RoboDK station: invisiblechess.rdk

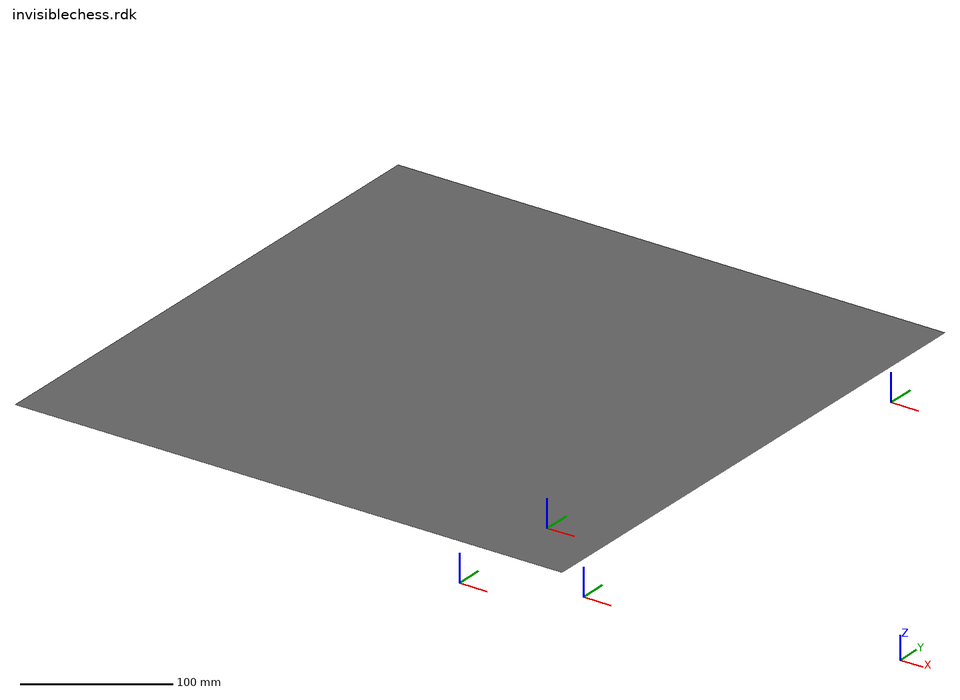
[picture v0: the station drawn from its stored meshes, robots at their saved joint values, targets as dots, program paths as lines]
Station invisiblechess (saved by RoboDK 5.6.5). Poses are relative to the parent item; angles as X-Y-Z fixed-axis rotations.
Station parameters (name, value as stored): Record_Record, 0
  - frame Frame 1 at (0, -100, 0) mm
    - object chessrobo at (100, -100, -10) mm, size 437.3 x 437.3 x 0 mm, 469029088 curves, geometry from chessrobo.png
    - object PAWN at (65, 300, -10) mm
    - object KNIGHT at (117, 146, -10) mm
    - object bishop at (-185, 150, -10) mm
    - object PAWN at (17, 96, -10) mm
    - object KNIGHT at (115, 300, -10) mm
    - object bishop at (17, 96, -10) mm
    - object PAWN at (67, 146, -10) mm
    - object KNIGHT at (-35, 200, -10) mm
    - object king at (67, 196, -10) mm
  - frame Frame 3 at (67, -54, -10) mm
    - object bishop at (0, 0, 0) mm
    - object PAWN at (0, 0, 0) mm
    - object ROOK at (-200, 0, 0) mm
    - object KNIGHT at (0, 0, 0) mm
    - object ROOK at (-200, 0, 0) mm
    - object PAWN at (0, 0, 0) mm
    - object PAWN at (0, 0, 0) mm
    - object PAWN at (0, 0, 0) mm
    - object PAWN at (0, 0, 0) mm
    - object QUEEN at (0, 0, 0) mm
    - object PAWN at (0, 0, 0) mm
  - Python program chess1 (listed below)
  - program rookie (3 instructions, listed below)
  - program backtobse (1 instructions, listed below)
  - frame Frame 4 at (0, 0, 0) mm
    - frame Frame 3 at (65, 300, -10) mm
      - object ROOK at (-200, 0, 0) mm
      - object king at (0, 0, 0) mm
      - object QUEEN at (0, 0, 0) mm
      - object ROOK at (-200, 0, 0) mm
      - object bishop at (0, 0, 0) mm
      - object PAWN at (0, 0, 0) mm
      - object PAWN at (0, 0, 0) mm
      - object PAWN at (0, 0, 0) mm
      - object PAWN at (0, 0, 0) mm
      - object PAWN at (0, 0, 0) mm
      - object PAWN at (0, 0, 0) mm
      - object PAWN at (0, 0, 0) mm
  - Python program Prog4 (listed below)
  - Python program chess (listed below)
  - program Prog6 (1 instructions, listed below)
  - program Prog7 (1 instructions, listed below)
  - program Prog8 (1 instructions, listed below)
  - program Prog9 (0 instructions, listed below)
  - program Prog10 (0 instructions, listed below)
  - Python program Prog11 (listed below)
  - Python program samattach (listed below)
  - Python program Prog13 (listed below)
  - Python program Prog14 (listed below)
  - Python program Prog15 (listed below)
  - Python program Prog16 (listed below)
  - frame My Mechanism Base at (0, 0, 0) mm
    - robot My Mechanism: 4 axes
        joint limits [-2000, -2000, -2000, -2000] to [2000, 2000, 2000, 2000]; home [0, 0, 0, 0]; saved at [-150, 150, -10, 0]
      - tool microagv1, TCP at (0, 0, 0) mm
  - Python program Prog17 (listed below)
  - Python program Prog18 (listed below)
  - Python program Prog19 (listed below)
  - Python program Prog20 (listed below)
  - Python program Prog21 (listed below)
  - Python program Prog22 (listed below)
  - Python program final (listed below)
  - Python program Prog24 (listed below)
  - Python program Prog25 (listed below)
  - frame Frame 6 at (-200, 150, 1000) mm, rotated rx 180 ry 0 rz -90 deg
    - camera Camera 1
  - Python program app (listed below)
  - Python program code (listed below)
  - Python program code (listed below)
  - Python program Prog29 (listed below)
  - frame Frame 7 at (0, 1150, 0) mm
  - Python program chessmaster1 (listed below)
  - Python program Prog31 (listed below)
  - Python program Prog32 (listed below)
  - Python program Prog33 (listed below)
  - Python program Prog34 (listed below)
  - Python program Prog35 (listed below)
  - Python program Prog36 (listed below)
  - Python program final (listed below)
  - Python program stockfish (listed below)
  - Python program RoboDKChessStockfishfinal (listed below)

--- Python program chess1 ---
# Type help("robodk.robolink") or help("robodk.robomath") for more information
# Press F5 to run the script
# Documentation: https://robodk.com/doc/en/RoboDK-API.html
# Reference:     https://robodk.com/doc/en/PythonAPI/robodk.html
# Note: It is not required to keep a copy of this file, your Python script is saved with your RDK project

# You can also use the new version of the API:
from robodk import robolink    # RoboDK API
from robodk import robomath    # Robot toolbox
RDK = robolink.Robolink()

# Forward and backwards compatible use of the RoboDK API:
# Remove these 2 lines to follow python programming guidelines
from robodk import *      # RoboDK API
from robolink import *    # Robot toolbox
# Link to RoboDK
# RDK = Robolink()

# Notify user:
print('To edit this program:\nright click on the Python program, then, select "Edit Python script"')

# Program example:

# Provoking an exception will display the console output if you run this script from RoboDK
#raise Exception('Program not edited.')
item = RDK.Item('My Mechanism')
if item.Valid():
    print('Item selected: ' + item.Name())
    print('Item position before move: ' + repr(item.Pose()))

def move_rook1():
    current_pose = item.Pose()
    new_pose = transl(-350, 0, 0) * current_pose
    item.MoveL(new_pose)

def move_rook2():
    current_pose = item.Pose()
    new_pose = transl(0, 350, 0) * current_pose
    item.MoveL(new_pose)

def move_rook3():
    current_pose = item.Pose()
    new_pose = transl(350, 0, 0) * current_pose
    item.MoveL(new_pose)

def move_rook4():
    current_pose = item.Pose()
    new_pose = transl(0, -350, 0) * current_pose
    item.MoveL(new_pose)

move_rook1()
move_rook2()
move_rook3()
move_rook4()

--- program rookie ---
  Attach to microagv1
  Call chess
  Detach from AGV

--- program backtobse ---
  Replace ROOK

--- Python program Prog4 ---
# Type help("robodk.robolink") or help("robodk.robomath") for more information
# Press F5 to run the script
# Documentation: https://robodk.com/doc/en/RoboDK-API.html
# Reference:     https://robodk.com/doc/en/PythonAPI/robodk.html
# Note: It is not required to keep a copy of this file, your Python script is saved with your RDK project

# You can also use the new version of the API:
from robodk import robolink    # RoboDK API
from robodk import robomath    # Robot toolbox
RDK = robolink.Robolink()

# Forward and backwards compatible use of the RoboDK API:
# Remove these 2 lines to follow python programming guidelines
from robodk import *      # RoboDK API
from robolink import *    # Robot toolbox
# Link to RoboDK
# RDK = Robolink()

# Notify user:
print('To edit this program:\nright click on the Python program, then, select "Edit Python script"')

# Program example:
item = RDK.Item('base')
if item.Valid():
    print('Item selected: ' + item.Name())
    print('Item posistion: ' + repr(item.Pose()))

print('Items in the station:')
itemlist = RDK.ItemList()
print(itemlist)

# Provoking an exception will display the console output if you run this script from RoboDK
#raise Exception('Program not edited.')
from robodk import robolink, transl

RDK = robolink.Robolink()

item = RDK.Item('My Mechanism')
if item.Valid():
    print('Item selected: ' + item.Name())
    print('Item position before move: ' + repr(item.Pose()))

# Define the grid and corresponding coordinates
grid_coordinates = {
    'a1': [0, 350, 0],
    'a2': [0, 300, 0],
    'a3': [-350, 350, 0],
    'a4': [-350, 700, 0],
    'a5': [-350, 1050, 0],
    'a6': [-350, 1400, 0],
    'a7': [-350, 1750, 0],
    'a8': [-350, 2100, 0],
    # Add similar entries for b1, c1, etc.
}

def move_to_square(square):
    if square in grid_coordinates:
        current_pose = item.Pose()
        new_pose = transl(*grid_coordinates[square]) * current_pose
        item.MoveL(new_pose)
    else:
        print(f"Square {square} not found in the grid_coordinates dictionary.")

# Prompt the user for input
#target_square = input("Enter the target square (e.g., a1, b3, h8): ")
#move_to_square(target_square)

while True:
    target_square = input("Enter the target square (e.g., a1, b3, h8) or 'no' to exit: ")

    if target_square.lower() == 'no':
        print("Exiting the program.")
        break  # Exit the loop if the user enters 'no'

    move_to_square(target_square)

--- Python program chess ---
from robodk import robolink    # RoboDK API
from robodk import robomath    # Robot toolbox
RDK = robolink.Robolink()

# Forward and backwards compatible use of the RoboDK API:
# Remove these 2 lines to follow python programming guidelines
from robodk import *      # RoboDK API
from robolink import *    # Robot toolbox
from robodk import robolink, transl
RDK = robolink.Robolink()

item = RDK.Item('My Mechanism')
tool = RDK.Item('AGV')
if item.Valid():
    print('Item selected: ' + item.Name())
    print('Item position before move: ' + repr(item.Pose()))
obj = RDK.Item('')
# Define the grid and corresponding coordinates
grid_coordinates = {
    'a1': [0, 350, -10],
    'a2': [0, 300, -10],
    'a3': [0, 250, -10],
    'a4': [0, 200, -10],
    'a5': [0, 150, -10],
    'a6': [0, 100, -10],
    'a7': [0, 50, -10],
    'a8': [0, 0, -10],
    'b1': [-50, 350, -10],
    'b2': [-50, 300, -10],
    'b3': [-50, 250, -10],
    'b4': [-50, 200, -10],
    'b5': [-50, 150, -10],
    'b6': [-50, 100, -10],
    'b7': [-50, 50, -10],
    'b8': [-50, 0, -10],
    'c1': [-100, 350, -10],
    'c2': [-100, 300, -10],
    'c3': [-100, 250, -10],
    'c4': [-100, 200, -10],
    'c5': [-100, 150, -10],
    'c6': [-100, 100, -10],
    'c7': [-100, 50, -10],
    'c8': [-100, 0, -10],
    'd1': [-150, 350, -10],
    'd2': [-150, 300, -10],
    'd3': [-150, 250, -10],
    'd4': [-150, 200, -10],
    'd5': [-150, 150, -10],
    'd6': [-150, 100, -10],
    'd7': [-150, 50, -10],
    'd8': [-150, 0, -10],
    'e1': [-200, 350, -10],
    'e2': [-200, 300, -10],
    'e3': [-200, 250, -10],
    'e4': [-200, 200, -10],
    'e5': [-200, 150, -10],
    'e6': [-200, 100, -10],
    'e7': [-200, 50, -10],
    'e8': [-200, 0, -10],
    'f1': [-250, 350, -10],
    'f2': [-250, 300, -10],
    'f3': [-250, 250, -10],
    'f4': [-250, 200, -10],
    'f5': [-250, 150, -10],
    'f6': [-250, 100, -10],
    'f7': [-250, 50, -10],
    'f8': [-250, 0, -10],
    'g1': [-300, 350, -10],
    'g2': [-300, 300, -10],
    'g3': [-300, 250, -10],
    'g4': [-300, 200, -10],
    'g5': [-300, 150, -10],
    'g6': [-300, 100, -10],
    'g7': [-300, 50, -10],
    'g8': [-300, 0, -10],
    'h1': [-350, 350, -10],
    'h2': [-350, 300, -10],
    'h3': [-350, 250, -10],
    'h4': [-350, 200, -10],
    'h5': [-350, 150, -10],
    'h6': [-350, 100, -10],
    'h7': [-350, 50, -10],
    'h8': [-350, 0, -10],
}

def move_to_square(square):
    if square in grid_coordinates:
        target_pose = transl(*grid_coordinates[square])
        item.setPose(target_pose)  # Set the robot's pose directly
    else:
        print(f"Square {square} not found in the grid_coordinates dictionary.")




# Loop to keep asking for input
while True:
    target_square = input("Enter the target square (e.g., a1, b3, h8) or 'no' to exit: ")

    if target_square.lower() == 'no':
        print("Exiting the program.")
        break  # Exit the loop if the user enters 'no'

    move_to_square(target_square)
    #tool.AttachClosest(list_objects=[obj])
    tool.RDK().RunProgram('Prog7')
    target_square = input("Enter the target square (e.g., a1, b3, h8) or 'no' to exit: ")

    if target_square.lower() == 'no':
        print("Exiting the program.")
        break  # Exit the loop if the user enters 'no'

    move_to_square(target_square)
    tool.RDK().RunProgram('Prog8')

--- program Prog6 ---
  Replace objects

--- program Prog7 ---
  Attach to microagv1

--- program Prog8 ---
  Detach from microagv1

--- program Prog9 ---

--- program Prog10 ---

--- Python program Prog11 ---
# Type help("robodk.robolink") or help("robodk.robomath") for more information
# Press F5 to run the script
# Documentation: https://robodk.com/doc/en/RoboDK-API.html
# Reference:     https://robodk.com/doc/en/PythonAPI/robodk.html
# Note: It is not required to keep a copy of this file, your Python script is saved with your RDK project

# You can also use the new version of the API:
from robodk import robolink    # RoboDK API
from robodk import robomath    # Robot toolbox
RDK = robolink.Robolink()

# Forward and backwards compatible use of the RoboDK API:
# Remove these 2 lines to follow python programming guidelines
from robodk import *      # RoboDK API
from robolink import *    # Robot toolbox
# Link to RoboDK
# RDK = Robolink()
from robodk import robolink, robomath
# Notify user:
print('To edit this program:\nright click on the Python program, then, select "Edit Python script"')

# Program example:
item = RDK.Item('My Mechanism')
if item.Valid():
    print('Item selected: ' + item.Name())
    print('Item posistion: ' + repr(item.Pose()))

print('Items in the station:')
itemlist = RDK.ItemList()
print(itemlist)

# Provoking an exception will display the console output if you run this script from RoboDK
#raise Exception('Program not edited.')
from robodk import robolink, transl
from robodk import robolink, robomath
RDK = robolink.Robolink()

# This will automatically select the robot if there is only one
robot = RDK.ItemUserPick("", robolink.ITEM_TYPE_ROBOT_ARM)
if not robot.Valid():
    quit()
RDK = robolink.Robolink()

item = RDK.Item('My Mechanism')
if item.Valid():
    print('Item selected: ' + item.Name())
    print('Item position before move: ' + repr(item.Pose()))

# Define the grid and corresponding coordinates
grid_coordinates = {
    'a1': [0, 350, 0],
    'a2': [0, 300, 0],
    'a3': [0, 250, 0],
    'a4': [0, 200, 0],
    'a5': [0, 150, 0],
    'a6': [0, 100, 0],
    'a7': [0, 50, 0],
    'a8': [0, 0, 0],
    # Add similar entries for b1, c1, etc.
}
# Retrieve the active tool of the robot
tool = RDK.getLink(robolink.ITEM_TYPE_TOOL)
if not tool.Valid():
    quit()

# Get the knight object and its current parent (to restore it later)
obj = RDK.Item('')
parent = obj.Parent()  # IMPORTANT! Parent must be a FRAME, not a folder..
def move_to_square(square):
    if square in grid_coordinates:
        target_pose = transl(*grid_coordinates[square])
        item.setPose(target_pose)  # Set the robot's pose directly

        # Attach the closest part on the first move
        closest_part = item.AttachClosest()
        if closest_part.Valid():
            print(f"Attached closest part: {closest_part.Name()}")

        # Detach on the second move
        second_move = input("Enter 'no' to exit or press Enter to make the second move: ")
        if second_move.lower() == 'no':
            print("Exiting the program.")
            return

        item.DetachAll()
        print("Detached all parts.")
    else:
        print(f"Square {square} not found in the grid_coordinates dictionary.")

# Loop to keep asking for input
while True:
    target_square = input("Enter the target square (e.g., a1, b3, h8) or 'no' to exit: ")

    if target_square.lower() == 'no':
        print("Exiting the program.")
        break  # Exit the loop if the user enters 'no'

    move_to_square(target_square)

--- Python program samattach ---
from robodk import robolink, robomath
RDK = robolink.Robolink()

# This will automatically select the robot if there is only one
robot = RDK.ItemUserPick("", robolink.ITEM_TYPE_ROBOT_ARM)
if not robot.Valid():
    quit()

# Retrieve the active tool of the robot
tool = robot.getLink(robolink.ITEM_TYPE_TOOL)
if not tool.Valid():
    quit()

# Get the knight object and its current parent (to restore it later)
obj = RDK.Item('KNIGHT W 1')
parent = obj.Parent() # IMPROTANT! Parent must be a FRAME, not a folder..

robot.MoveJ(RDK.Item('App Pick'))
robot.MoveL(RDK.Item('Pick'))

# In Tools-Options-Station -> check "Check shorted distance between TCP and object shape"
tool.AttachClosest(list_objects=[obj])

robot.MoveL(RDK.Item('App Pick'))
robomath.pause(2)
robot.MoveL(RDK.Item('Pick'))
tool.DetachAll(parent)
robot.MoveL(RDK.Item('App Pick'))

--- Python program Prog13 ---
# Type help("robodk.robolink") or help("robodk.robomath") for more information
# Press F5 to run the script
# Documentation: https://robodk.com/doc/en/RoboDK-API.html
# Reference:     https://robodk.com/doc/en/PythonAPI/robodk.html
# Note: It is not required to keep a copy of this file, your Python script is saved with your RDK project

# You can also use the new version of the API:
from robodk import robolink    # RoboDK API
from robodk import robomath    # Robot toolbox
RDK = robolink.Robolink()

# Forward and backwards compatible use of the RoboDK API:
# Remove these 2 lines to follow python programming guidelines
from robodk import *      # RoboDK API
from robolink import *    # Robot toolbox
# Link to RoboDK
# RDK = Robolink()

# Notify user:
print('To edit this program:\nright click on the Python program, then, select "Edit Python script"')

# Program example:
item = RDK.Item('base')
if item.Valid():
    print('Item selected: ' + item.Name())
    print('Item posistion: ' + repr(item.Pose()))

print('Items in the station:')
itemlist = RDK.ItemList()
print(itemlist)

# Provoking an exception will display the console output if you run this script from RoboDK
raise Exception('Program not edited.')

--- Python program Prog14 ---
from robodk import robolink, ITEM_TYPE_ROBOT_ARM

RDK = robolink.Robolink()

# Retrieve the robot if there is only one
robot = RDK.ItemUserPick("Select a robot", ITEM_TYPE_ROBOT_ARM)
if not robot.Valid():
    quit()

# Retrieve the active tool of the robot
tool = robot.Child()
if not tool.Valid():
    quit()

# Define the grid and corresponding coordinates
grid_coordinates = {
    'a1': [0, 350, 0],
    'a2': [0, 300, 0],
    'a3': [0, 250, 0],
    'a4': [0, 200, 0],
    'a5': [0, 150, 0],
    'a6': [0, 100, 0],
    'a7': [0, 50, 0],
    'a8': [0, 0, 0],
    # Add similar entries for b1, c1, etc.
}

def move_to_square(square):
    if square in grid_coordinates:
        target_pose = robolink.transl(*grid_coordinates[square])
        robot.setPose(target_pose)  # Set the robot's pose directly
        return True
    else:
        print(f"Square {square} not found in the grid_coordinates dictionary.")
        return False

# Variables to keep track of the state
attached = False

# Loop to keep asking for input
while True:
    target_square = input("Enter the target square (e.g., a1, b3, h8) or 'no' to exit: ")

    if target_square.lower() == 'no':
        print("Exiting the program.")
        break  # Exit the loop if the user enters 'no'

    if attached:
        tool.DetachAll()
        print("Detached part.")
        attached = False
    else:
        success = move_to_square(target_square)
        if success:
            tool.AttachClosest()
            print("Attached closest part.")
            attached = True

--- Python program Prog15 ---
# Type help("robodk.robolink") or help("robodk.robomath") for more information
# Press F5 to run the script
# Documentation: https://robodk.com/doc/en/RoboDK-API.html
# Reference:     https://robodk.com/doc/en/PythonAPI/robodk.html
# Note: It is not required to keep a copy of this file, your Python script is saved with your RDK project

# You can also use the new version of the API:
from robodk import robolink    # RoboDK API
from robodk import robomath    # Robot toolbox
RDK = robolink.Robolink()

# Forward and backwards compatible use of the RoboDK API:
# Remove these 2 lines to follow python programming guidelines
from robodk import *      # RoboDK API
from robolink import *    # Robot toolbox
# Link to RoboDK
# RDK = Robolink()

# Notify user:
print('To edit this program:\nright click on the Python program, then, select "Edit Python script"')

# Program example:
item = RDK.Item('base')
if item.Valid():
    print('Item selected: ' + item.Name())
    print('Item posistion: ' + repr(item.Pose()))

print('Items in the station:')
itemlist = RDK.ItemList()
print(itemlist)

# Provoking an exception will display the console output if you run this script from RoboDK
#raise Exception('Program not edited.')
from robodk import *

RDK = robolink.Robolink()

# Retrieve the robot if there is only one
robot = RDK.ItemUserPick("Select a robot", ITEM_TYPE_ROBOT_ARM)
if not robot.Valid():
    quit()

# Retrieve the active tool of the robot
tool = robot.Child()
if not tool.Valid():
    quit()

# Define the grid and corresponding coordinates
grid_coordinates = {
    'a1': [0, 350, 0],
    'a2': [0, 300, 0],
    'a3': [0, 250, 0],
    'a4': [0, 200, 0],
    'a5': [0, 150, 0],
    'a6': [0, 100, 0],
    'a7': [0, 50, 0],
    'a8': [0, 0, 0],
    # Add similar entries for b1, c1, etc.
}

def move_to_square(square):
    if square in grid_coordinates:
        target_pose = transl(*grid_coordinates[square])
        robot.setPose(target_pose)  # Set the robot's pose directly
        return True
    else:
        print(f"Square {square} not found in the grid_coordinates dictionary.")
        return False

# Variables to keep track of the state
attached = False

# Loop to keep asking for input
while True:
    target_square = input("Enter the target square (e.g., a1, b3, h8) or 'no' to exit: ")

    if target_square.lower() == 'no':
        print("Exiting the program.")
        break  # Exit the loop if the user enters 'no'

    if attached:
        tool.DetachAll()
        print("Detached part.")
        attached = False
    else:
        success = move_to_square(target_square)
        if success:
            tool.AttachClosest()
            print("Attached closest part.")
            attached = True

--- Python program Prog16 ---
# Type help("robodk.robolink") or help("robodk.robomath") for more information
# Press F5 to run the script
# Documentation: https://robodk.com/doc/en/RoboDK-API.html
# Reference:     https://robodk.com/doc/en/PythonAPI/robodk.html
# Note: It is not required to keep a copy of this file, your Python script is saved with your RDK project

# You can also use the new version of the API:
from robodk import robolink    # RoboDK API
from robodk import robomath    # Robot toolbox
RDK = robolink.Robolink()

# Forward and backwards compatible use of the RoboDK API:
# Remove these 2 lines to follow python programming guidelines
from robodk import *      # RoboDK API
from robolink import *    # Robot toolbox
# Link to RoboDK
# RDK = Robolink()

# Notify user:
print('To edit this program:\nright click on the Python program, then, select "Edit Python script"')

# Program example:
item = RDK.Item('base')
if item.Valid():
    print('Item selected: ' + item.Name())
    print('Item posistion: ' + repr(item.Pose()))

print('Items in the station:')
itemlist = RDK.ItemList()
print(itemlist)

# Provoking an exception will display the console output if you run this script from RoboDK
#raise Exception('Program not edited.')
from robodk import robolink, transl
import chess
import chess.engine

RDK = robolink.Robolink()

item = RDK.Item('My Mechanism')
tool = RDK.Item('AGV')
if item.Valid():
    print('Item selected: ' + item.Name())
    print('Item position before move: ' + repr(item.Pose()))
obj = RDK.Item('')
# Define the grid and corresponding coordinates
grid_coordinates = {
    'a1': [0, 350, 10],
    'a2': [0, 300, 10],
    'a3': [0, 250, 10],
    'a4': [0, 200, 10],
    'a5': [0, 150, 10],
    'a6': [0, 100, 10],
    'a7': [0, 50, 10],
    'a8': [0, 0, 10],
    # Add similar entries for b1, c1, etc.
}

def move_to_square(square):
    if square in grid_coordinates:
        target_pose = transl(*grid_coordinates[square])
        item.setPose(target_pose)  # Set the robot's pose directly
    else:
        print(f"Square {square} not found in the grid_coordinates dictionary.")

def stockfish_move(board):
    with chess.engine.SimpleEngine.popen_uci("/path/to/stockfish") as engine:
        result = engine.play(board, chess.engine.Limit(time=2.0))
        return result.move

# Loop to keep asking for input
while True:
    target_square = input("Enter the target square (e.g., a1, b3, h8) or 'no' to exit: ")

    if target_square.lower() == 'no':
        print("Exiting the program.")
        break  # Exit the loop if the user enters 'no'

    move_to_square(target_square)
    tool.RDK().RunProgram('Prog7')

    board = chess.Board()
    opponent_move = stockfish_move(board)
    print("Opponent's move:", opponent_move.uci())

    # Assuming opponent_move.uci() returns a valid square (e.g., "e2e4")
    move_to_square(opponent_move.uci())
    tool.RDK().RunProgram('Prog8')

--- Python program Prog17 ---
# Type help("robodk.robolink") or help("robodk.robomath") for more information
# Press F5 to run the script
# Documentation: https://robodk.com/doc/en/RoboDK-API.html
# Reference:     https://robodk.com/doc/en/PythonAPI/robodk.html
# Note: It is not required to keep a copy of this file, your Python script is saved with your RDK project

# You can also use the new version of the API:
from robodk import robolink    # RoboDK API
from robodk import robomath    # Robot toolbox
RDK = robolink.Robolink()

# Forward and backwards compatible use of the RoboDK API:
# Remove these 2 lines to follow python programming guidelines
from robodk import *      # RoboDK API
from robolink import *    # Robot toolbox
# Link to RoboDK
# RDK = Robolink()

# Notify user:
print('To edit this program:\nright click on the Python program, then, select "Edit Python script"')

# Program example:
item = RDK.Item('base')
if item.Valid():
    print('Item selected: ' + item.Name())
    print('Item posistion: ' + repr(item.Pose()))

print('Items in the station:')
itemlist = RDK.ItemList()
print(itemlist)

# Provoking an exception will display the console output if you run this script from RoboDK
#raise Exception('Program not edited.')
import chess
from serial.tools import list_ports
#import chess.svg
import chess.engine
def main():
    # Specify the full path to your Stockfish executable
    engine_path = "stockfish\stockfish-windows-x86-64-avx2"  # Replace with the actual name of your Stockfish executable

    # Create a Chess engine with Stockfish
    engine = chess.engine.SimpleEngine.popen_uci(engine_path)

    board = chess.Board()

--- Python program Prog18 ---
# Type help("robodk.robolink") or help("robodk.robomath") for more information
# Press F5 to run the script
# Documentation: https://robodk.com/doc/en/RoboDK-API.html
# Reference:     https://robodk.com/doc/en/PythonAPI/robodk.html
# Note: It is not required to keep a copy of this file, your Python script is saved with your RDK project

# You can also use the new version of the API:
from robodk import robolink    # RoboDK API
from robodk import robomath    # Robot toolbox
RDK = robolink.Robolink()

# Forward and backwards compatible use of the RoboDK API:
# Remove these 2 lines to follow python programming guidelines
from robodk import *      # RoboDK API
from robolink import *    # Robot toolbox
# Link to RoboDK
# RDK = Robolink()

# Notify user:
#print('To edit this program:\nright click on the Python program, then, select "Edit Python script"')

# Program example:
item = RDK.Item('base')
if item.Valid():
    print('Item selected: ' + item.Name())
    print('Item posistion: ' + repr(item.Pose()))

print('Items in the station:')
itemlist = RDK.ItemList()
#print(itemlist)

# Provoking an exception will display the console output if you run this script from RoboDK
#raise Exception('Program not edited.')
from robolink import import_install
import_install("chess")
import chess
from robolink import import_install
import_install("stockfish")
import stockfish
from stockfish import Stockfish

stockfish = Stockfish(path= "/Users/dancr/chess-robot/stockfish/stockfish-windows-x86-64-avx2.exe")
boardmac = stockfish.get_board_visual()
boardmaco = stockfish.get_best_move()
print(boardmac)
print(boardmaco)

--- Python program Prog19 ---
# Type help("robodk.robolink") or help("robodk.robomath") for more information
# Press F5 to run the script
# Documentation: https://robodk.com/doc/en/RoboDK-API.html
# Reference:     https://robodk.com/doc/en/PythonAPI/robodk.html
# Note: It is not required to keep a copy of this file, your Python script is saved with your RDK project

# You can also use the new version of the API:
from robodk import robolink    # RoboDK API
from robodk import robomath    # Robot toolbox
RDK = robolink.Robolink()

# Forward and backwards compatible use of the RoboDK API:
# Remove these 2 lines to follow python programming guidelines
from robodk import *      # RoboDK API
from robolink import *    # Robot toolbox
# Link to RoboDK
# RDK = Robolink()

# Notify user:
print('To edit this program:\nright click on the Python program, then, select "Edit Python script"')

# Program example:
item = RDK.Item('base')
if item.Valid():
    print('Item selected: ' + item.Name())
    print('Item posistion: ' + repr(item.Pose()))

print('Items in the station:')
itemlist = RDK.ItemList()
print(itemlist)

# Provoking an exception will display the console output if you run this script from RoboDK
#raise Exception('Program not edited.')
from robodk import robolink
from robolink import import_install
from stockfish import Stockfish

# Initialize RoboDK
RDK = robolink.Robolink()

# Install chess and stockfish libraries
import_install("chess")
import chess
import_install("stockfish")
import stockfish

# Initialize Stockfish
stockfish = Stockfish(path="/Users/dancr/chess-robot/stockfish/stockfish-windows-x86-64-avx2.exe")

# Get the best move suggestion from Stockfish
best_move = stockfish.get_best_move()

# Parse the move suggestion
try:
    move = chess.Move.from_uci(best_move)
    starting_square = chess.square_name(move.from_square)
    ending_square = chess.square_name(move.to_square)

    print("Starting Square:", starting_square)
    print("Ending Square:", ending_square)

except ValueError as e:
    print("Error parsing move suggestion:", e)
board_visual = stockfish.get_board_visual()
print(board_visual)
stockfish.set_position([best_move])
board_visual = stockfish.get_board_visual()
print(board_visual)

--- Python program Prog20 ---
# Type help("robodk.robolink") or help("robodk.robomath") for more information
# Press F5 to run the script
# Documentation: https://robodk.com/doc/en/RoboDK-API.html
# Reference:     https://robodk.com/doc/en/PythonAPI/robodk.html
# Note: It is not required to keep a copy of this file, your Python script is saved with your RDK project

# You can also use the new version of the API:
from robodk import robolink    # RoboDK API
from robodk import robomath    # Robot toolbox
RDK = robolink.Robolink()

# Forward and backwards compatible use of the RoboDK API:
# Remove these 2 lines to follow python programming guidelines
from robodk import *      # RoboDK API
from robolink import *    # Robot toolbox
# Link to RoboDK
# RDK = Robolink()

# Notify user:
print('To edit this program:\nright click on the Python program, then, select "Edit Python script"')

# Program example:
item = RDK.Item('base')
if item.Valid():
    print('Item selected: ' + item.Name())
    print('Item posistion: ' + repr(item.Pose()))

#print('Items in the station:')
itemlist = RDK.ItemList()
#print(itemlist)

# Provoking an exception will display the console output if you run this script from RoboDK
#raise Exception('Program not edited.')
from robodk import robolink
from robolink import import_install
from stockfish import Stockfish
import chess

# Initialize RoboDK
RDK = robolink.Robolink()

# Install chess and stockfish libraries
import_install("chess")
import chess
import_install("stockfish")
import stockfish

# Initialize Stockfish
stockfish = Stockfish(path="/Users/dancr/chess-robot/stockfish/stockfish-windows-x86-64-avx2.exe")

# Function to update the board and get user's move
def play_chess():
    while True:
        # Get the best move suggestion from Stockfish
        best_move = stockfish.get_best_move()
        print(best_move)

        # Parse the move suggestion
        try:
            move = chess.Move.from_uci(best_move)
            starting_square = chess.square_name(move.from_square)
            ending_square = chess.square_name(move.to_square)

            print("Stockfish suggests move:")
            print("Starting Square:", starting_square)
            print("Ending Square:", ending_square)

            # Update the board with Stockfish's move
            stockfish.set_position([best_move])
            board_visual = stockfish.get_board_visual()
            print(board_visual)

            # Ask user for their move in UCI format
            user_move = input("Enter your move (UCI format): ")

            # Update the board with the user's move
            stockfish.set_position([user_move])
            board_visual = stockfish.get_board_visual()
            print(board_visual)

        except ValueError as e:
            print("Error parsing move suggestion:", e)
            break

# Start the chess game
play_chess()

--- Python program Prog21 ---
# Type help("robodk.robolink") or help("robodk.robomath") for more information
# Press F5 to run the script
# Documentation: https://robodk.com/doc/en/RoboDK-API.html
# Reference:     https://robodk.com/doc/en/PythonAPI/robodk.html
# Note: It is not required to keep a copy of this file, your Python script is saved with your RDK project

# You can also use the new version of the API:
from robodk import robolink    # RoboDK API
from robodk import robomath    # Robot toolbox
RDK = robolink.Robolink()

# Forward and backwards compatible use of the RoboDK API:
# Remove these 2 lines to follow python programming guidelines
from robodk import *      # RoboDK API
from robolink import *    # Robot toolbox
# Link to RoboDK
# RDK = Robolink()

# Notify user:
print('To edit this program:\nright click on the Python program, then, select "Edit Python script"')

# Program example:
item = RDK.Item('base')
if item.Valid():
    print('Item selected: ' + item.Name())
    print('Item posistion: ' + repr(item.Pose()))

#print('Items in the station:')
itemlist = RDK.ItemList()
#print(itemlist)

# Provoking an exception will display the console output if you run this script from RoboDK
#raise Exception('Program not edited.')
from robodk import robolink
#from robodk import import_install
from stockfish import Stockfish
#import chess

# Initialize RoboDK
RDK = robolink.Robolink()


# Initialize Stockfish
stockfish = Stockfish(path="/Users/dancr/chess-robot/stockfish/stockfish-windows-x86-64-avx2.exe")

# Function to update the board and get user's move
def play_chess():
    while True:
        # Get the best move suggestion from Stockfish
        best_move = stockfish.get_best_move()

        # Parse the move suggestion
        try:
            move = chess.Move.from_uci(best_move)
            starting_square = chess.square_name(move.from_square)
            ending_square = chess.square_name(move.to_square)

            print("Stockfish suggests move:")
            print("Starting Square:", starting_square)
            print("Ending Square:", ending_square)

            # Update the board with Stockfish's move
            stockfish.set_position([best_move])
            board_visual = stockfish.get_board_visual()
            print(board_visual)

            # Ask user for their move in UCI format
            user_move = input("Enter your move (UCI format, e.g., e7e5): ")

            # Validate and update the board with the user's move
            try:
                user_move_obj = chess.Move.from_uci(user_move)
                if user_move_obj in chess.Board(board_visual).legal_moves:
                    stockfish.set_position([user_move])
                    board_visual = stockfish.get_board_visual()
                    print(board_visual)
                else:
                    print("Invalid move. Please enter a legal move.")
            except ValueError as e:
                print("Error parsing user's move:", e)

        except ValueError as e:
            print("Error parsing move suggestion:", e)
            break

# Start the chess game
play_chess()

--- Python program Prog22 ---
# Type help("robodk.robolink") or help("robodk.robomath") for more information
# Press F5 to run the script
# Documentation: https://robodk.com/doc/en/RoboDK-API.html
# Reference:     https://robodk.com/doc/en/PythonAPI/robodk.html
# Note: It is not required to keep a copy of this file, your Python script is saved with your RDK project

# You can also use the new version of the API:
from robodk import robolink    # RoboDK API
from robodk import robomath    # Robot toolbox
RDK = robolink.Robolink()

# Forward and backwards compatible use of the RoboDK API:
# Remove these 2 lines to follow python programming guidelines
from robodk import *      # RoboDK API
from robolink import *    # Robot toolbox
# Link to RoboDK
# RDK = Robolink()

# Notify user:
print('To edit this program:\nright click on the Python program, then, select "Edit Python script"')

# Program example:
item = RDK.Item('base')
if item.Valid():
    print('Item selected: ' + item.Name())
    print('Item posistion: ' + repr(item.Pose()))

#print('Items in the station:')
itemlist = RDK.ItemList()
#print(itemlist)

# Provoking an exception will display the console output if you run this script from RoboDK
#raise Exception('Program not edited.')
from robodk import robolink
#from robodk import import_install
from stockfish import Stockfish
import chess

# Initialize RoboDK
RDK = robolink.Robolink()

# Install chess and stockfish libraries
import_install("chess")
import chess
import_install("stockfish")
import stockfish

# Initialize Stockfish
stockfish = Stockfish(path="/Users/dancr/chess-robot/stockfish/stockfish-windows-x86-64-avx2.exe")

# Function to update the board and get user's move
def play_chess():
    while True:
        # Get the best move suggestion from Stockfish
        best_move = stockfish.get_best_move()

        # Parse the move suggestion
        try:
            move = chess.Move.from_uci(best_move)
            starting_square = chess.square_name(move.from_square)
            ending_square = chess.square_name(move.to_square)

            print("Stockfish suggests move:")
            print("Starting Square:", starting_square)
            print("Ending Square:", ending_square)

            # Update the board with Stockfish's move
            stockfish.set_position([best_move])
            board_visual = stockfish.get_board_visual()
            print(board_visual)

            # Ask user for their move in UCI format
            user_move = input("Enter your move (UCI format, e.g., e7e5): ")

            # Validate and update the board with the user's move
            try:
                stockfish.make_moves_from_current_position([user_move])
                board_visual = stockfish.get_board_visual()
                print(board_visual)
            except ValueError as e:
                print("Error making user's move:", e)

        except ValueError as e:
            print("Error parsing move suggestion:", e)
            break

# Start the chess game
play_chess()

--- Python program final ---
# Type help("robodk.robolink") or help("robodk.robomath") for more information
# Press F5 to run the script
# Documentation: https://robodk.com/doc/en/RoboDK-API.html
# Reference:     https://robodk.com/doc/en/PythonAPI/robodk.html
# Note: It is not required to keep a copy of this file, your Python script is saved with your RDK project

# You can also use the new version of the API:
from robodk import robolink    # RoboDK API
from robodk import robomath    # Robot toolbox
RDK = robolink.Robolink()

# Forward and backwards compatible use of the RoboDK API:
# Remove these 2 lines to follow python programming guidelines
from robodk import *      # RoboDK API
from robolink import *    # Robot toolbox
# Link to RoboDK
# RDK = Robolink()

# Notify user:
print('To edit this program:\nright click on the Python program, then, select "Edit Python script"')

# Program example:
item = RDK.Item('base')
if item.Valid():
    print('Item selected: ' + item.Name())
    print('Item posistion: ' + repr(item.Pose()))

#print('Items in the station:')
itemlist = RDK.ItemList()
#print(itemlist)

# Provoking an exception will display the console output if you run this script from RoboDK
#raise Exception('Program not edited.')
#from robodk import robolink
#from robodk import import_install
from stockfish import Stockfish
import chess

# Initialize RoboDK
RDK = robolink.Robolink()

# Install chess and stockfish libraries
#import_install("chess")
import chess
#import_install("stockfish")
import stockfish

# Initialize Stockfish
stockfish = Stockfish(path="/Users/dancr/chess-robot/stockfish/stockfish-windows-x86-64-avx2.exe")

# Function to update the board and get user's move
def play_chess():
    while True:
        # Get the best move suggestion from Stockfish
        best_move = stockfish.get_best_move()

        # Parse the move suggestion
        try:
            move = chess.Move.from_uci(best_move)
            starting_square = chess.square_name(move.from_square)
            ending_square = chess.square_name(move.to_square)

            print("Stockfish suggests move:")
            print("Starting Square:", starting_square)
            print("Ending Square:", ending_square)

            # Ask user for their move in UCI format
            user_move = input("Enter your move (UCI format, e.g., e7e5): ")

            # Validate and update the board with Stockfish's and user's move
            try:
                stockfish.make_moves_from_current_position([best_move, user_move])
                board_visual = stockfish.get_board_visual()
                print(board_visual)
            except ValueError as e:
                print("Error making moves:", e)

        except ValueError as e:
            print("Error parsing move suggestion:", e)
            break

# Start the chess game
play_chess()

--- Python program Prog24 ---
# Type help("robodk.robolink") or help("robodk.robomath") for more information
# Press F5 to run the script
# Documentation: https://robodk.com/doc/en/RoboDK-API.html
# Reference:     https://robodk.com/doc/en/PythonAPI/robodk.html
# Note: It is not required to keep a copy of this file, your Python script is saved with your RDK project

# You can also use the new version of the API:
from robodk import robolink    # RoboDK API
from robodk import robomath    # Robot toolbox
RDK = robolink.Robolink()

# Forward and backwards compatible use of the RoboDK API:
# Remove these 2 lines to follow python programming guidelines
from robodk import *      # RoboDK API
from robolink import *    # Robot toolbox
# Link to RoboDK
# RDK = Robolink()

# Notify user:
print('To edit this program:\nright click on the Python program, then, select "Edit Python script"')

# Program example:
item = RDK.Item('base')
if item.Valid():
    print('Item selected: ' + item.Name())
    print('Item posistion: ' + repr(item.Pose()))

#print('Items in the station:')
#itemlist = RDK.ItemList()
#print(itemlist)

# Provoking an exception will display the console output if you run this script from RoboDK
#raise Exception('Program not edited.')
import chess
import chess.svg
import chess.engine

# Initialize the chess board
board = chess.Board()

# Function to print the current board
#def print_board(board):
    #display(chess.svg.board(board=board))

# Function to get legal moves for a given position
def get_legal_moves(board):
    legal_moves = list(board.legal_moves)
    return legal_moves

# Function to play a move and update the board
def play_move(board, move):
    if move in board.legal_moves:
        board.push(move)
    else:
        print("Invalid move!")

# Function to get Stockfish's suggested move
def get_stockfish_move(board, depth=20):
    with chess.engine.SimpleEngine.popen_uci("Users\dancr\chess-robot\stockfish\stockfish-windows-x86-64-avx2") as engine:
        result = engine.play(board, chess.engine.Limit(depth=depth))
        return result.move

# Main game loop
while not board.is_game_over():
    #print_board(board)
    print("Legal moves:", get_legal_moves(board))

    # Get player input
    move_input = input("Enter your move (e.g., 'a2a3'): ")

    # Parse player's move
    try:
        move = chess.Move.from_uci(move_input)
        play_move(board, move)
    except ValueError:
        print("Invalid move format! Use UCI notation (e.g., 'a2a3')")
        continue

    # Get Stockfish's move
    stockfish_move = get_stockfish_move(board)
    play_move(board, stockfish_move)

print("Game Over")

--- Python program Prog25 ---
# Type help("robodk.robolink") or help("robodk.robomath") for more information
# Press F5 to run the script
# Documentation: https://robodk.com/doc/en/RoboDK-API.html
# Reference:     https://robodk.com/doc/en/PythonAPI/robodk.html
# Note: It is not required to keep a copy of this file, your Python script is saved with your RDK project

# You can also use the new version of the API:
from robodk import robolink    # RoboDK API
from robodk import robomath    # Robot toolbox
RDK = robolink.Robolink()

# Forward and backwards compatible use of the RoboDK API:
# Remove these 2 lines to follow python programming guidelines
from robodk import *      # RoboDK API
from robolink import *    # Robot toolbox
# Link to RoboDK
# RDK = Robolink()

# Notify user:
print('To edit this program:\nright click on the Python program, then, select "Edit Python script"')

# Program example:
item = RDK.Item('base')
if item.Valid():
    print('Item selected: ' + item.Name())
    print('Item posistion: ' + repr(item.Pose()))

#print('Items in the station:')
itemlist = RDK.ItemList()
#print(itemlist)

# Provoking an exception will display the console output if you run this script from RoboDK
#raise Exception('Program not edited.')
from robodk import robolink
from stockfish import Stockfish
import chess

# Initialize RoboDK
RDK = robolink.Robolink()

# Install chess and stockfish libraries
import chess
import stockfish

# Initialize Stockfish
stockfish = Stockfish(path="/Users/dancr/chess-robot/stockfish/stockfish-windows-x86-64-avx2.exe")

# Function to update the board and get user's move
def play_chess():
    while True:
        # Get the best move suggestion from Stockfish
        best_move = stockfish.get_best_move()

        # Parse the move suggestion
        try:
            move = chess.Move.from_uci(best_move)
            starting_square = chess.square_name(move.from_square)
            ending_square = chess.square_name(move.to_square)

            print("Stockfish suggests move:")
            print("Starting Square:", starting_square)
            print("Ending Square:", ending_square)

            # Ask user for their move in UCI format
            user_move = input("Enter your move (UCI format, e.g., e7e5): ")

            # Validate and update the board with Stockfish's and user's move
            try:
                stockfish.make_moves_from_current_position([best_move, user_move])
                board_visual = stockfish.get_board_visual()
                print(board_visual)
            except ValueError as e:
                print("Error making moves:", e)

        except ValueError as e:
            print("Error parsing move suggestion:", e)
            break

# Start the chess game
play_chess()

--- Python program app ---
import tkinter as tk
from tkinter import ttk


def greet():
    print("a1")


root = tk.Tk()
root.title("a1")

greet_button = ttk.Button(root, text="a1", command=greet)
greet_button.pack(side="left", fill="x", expand=True)

quit_button = ttk.Button(root, text="Quit", command=root.destroy)
quit_button.pack(side="left", fill="x", expand=True)  # could use side="right"

root.mainloop()

--- Python program code ---
import tkinter as tk
from tkinter import ttk

# -- Windows only configuration --
try:
    from ctypes import windll
    windll.shcore.SetProcessDpiAwareness(1)
except:
    pass
# -- End Windows only configuration --

root = tk.Tk()
root.resizable(False, False)
root.title("Widget Examples")

# -- Text widgets --

# height is the number of rows of text
text = tk.Text(root, height=8)  # Show what happens if you `.pack()` here, while still assigning to variable.
text.pack()

# Insert content into the text area
text.insert("1.0", "Please enter a comment...")  # Can use \n to insert multiple lines.

# First argument: position within textarea.
# Second argument: text to insert after that position.

# The position is given as two numbers, separated by a `.`.
# First number is the line number, starting at 1.
# Second number is character number within the line, starting at 0.
# So 1.0 is the first line, first character.

# -- Disable text widget --

text["state"] = "disabled"  # "normal" is the counterpart

# -- Get text content --

text_content = text.get("1.0", "end")
print(text_content)

root.mainloop()

--- Python program code ---
import tkinter as tk
from tkinter import ttk


root = tk.Tk()
style = ttk.Style(root)

style.theme_use("clam")

style.map("CustomButton.TButton",
    foreground=[('pressed', 'red'), ('active', 'white')],
    background=[('pressed', '!disabled', 'black'), ('active', 'black')],  # Note that background colour can't be changed in the default Windows theme.
    font=[("pressed", ("TkDefaultFont", 15))]  # This may not make sense, but it still works
)

name = ttk.Label(root, text="Hello, world!")
entry = ttk.Entry(root, width=15)
button = ttk.Button(root, text="Press me.", style="CustomButton.TButton")
name.pack()
entry.pack()
button.pack()


root.mainloop()

--- Python program Prog29 ---
import tkinter as tk

def on_square_click(square):
    print("Selected square:", square)

root = tk.Tk()
root.title("Chessboard")

# Function to create a button with given row and column
def create_button(row, col):
    square = chr(ord('a') + col) + str(8 - row)
    button = tk.Button(root, text=square, width=3, height=1, command=lambda: on_square_click(square))
    button.grid(row=row, column=col, padx=2, pady=2)

# Create 8x8 grid of buttons
for row in range(8):
    for col in range(8):
        create_button(row, col)

root.mainloop()

--- Python program chessmaster1 ---
# Type help("robodk.robolink") or help("robodk.robomath") for more information
# Press F5 to run the script
# Documentation: https://robodk.com/doc/en/RoboDK-API.html
# Reference:     https://robodk.com/doc/en/PythonAPI/robodk.html
# Note: It is not required to keep a copy of this file, your Python script is saved with your RDK project

# You can also use the new version of the API:
from robodk import robolink    # RoboDK API
from robodk import robomath    # Robot toolbox
RDK = robolink.Robolink()

# Forward and backwards compatible use of the RoboDK API:
# Remove these 2 lines to follow python programming guidelines
from robodk import *      # RoboDK API
from robolink import *    # Robot toolbox
# Link to RoboDK
# RDK = Robolink()

#import chess

#import chess.engine
#board = chess.Board
# Notify user:
#print('To edit this program:\nright click on the Python program, then, select "Edit Python script"')

# Program example:

# Provoking an exception will display the console output if you run this script from RoboDK
#raise Exception('Program not edited.')
from robodk import robolink, transl
RDK = robolink.Robolink()
# This will automatically select the robot if there is only one


item = RDK.Item('My Mechanism')
tool = RDK.Item('AGV')
if item.Valid():
    print('Item selected: ' + item.Name())
    print('Item position before move: ' + repr(item.Pose()))
obj = RDK.Item('')
# Define the grid and corresponding coordinates
grid_coordinates = {
    'a1': [0, 350, -10],
    'a2': [0, 300, -10],
    'a3': [0, 250, -10],
    'a4': [0, 200, -10],
    'a5': [0, 150, -10],
    'a6': [0, 100, -10],
    'a7': [0, 50, -10],
    'a8': [0, 0, -10],
    'b1': [-50, 350, -10],
    'b2': [-50, 300, -10],
    'b3': [-50, 250, -10],
    'b4': [-50, 200, -10],
    'b5': [-50, 150, -10],
    'b6': [-50, 100, -10],
    'b7': [-50, 50, -10],
    'b8': [-50, 0, -10],
    'c1': [-100, 350, -10],
    'c2': [-100, 300, -10],
    'c3': [-100, 250, -10],
    'c4': [-100, 200, -10],
    'c5': [-100, 150, -10],
    'c6': [-100, 100, -10],
    'c7': [-100, 50, -10],
    'c8': [-100, 0, -10],
    'd1': [-150, 350, -10],
    'd2': [-150, 300, -10],
    'd3': [-150, 250, -10],
    'd4': [-150, 200, -10],
    'd5': [-150, 150, -10],
    'd6': [-150, 100, -10],
    'd7': [-150, 50, -10],
    'd8': [-150, 0, -10],
    'e1': [-200, 350, -10],
    'e2': [-200, 300, -10],
    'e3': [-200, 250, -10],
    'e4': [-200, 200, -10],
    'e5': [-200, 150, -10],
    'e6': [-200, 100, -10],
    'e7': [-200, 50, -10],
    'e8': [-200, 0, -10],
    'f1': [-250, 350, -10],
    'f2': [-250, 300, -10],
    'f3': [-250, 250, -10],
    'f4': [-250, 200, -10],
    'f5': [-250, 150, -10],
    'f6': [-250, 100, -10],
    'f7': [-250, 50, -10],
    'f8': [-250, 0, -10],
    'g1': [-300, 350, -10],
    'g2': [-300, 300, -10],
    'g3': [-300, 250, -10],
    'g4': [-300, 200, -10],
    'g5': [-300, 150, -10],
    'g6': [-300, 100, -10],
    'g7': [-300, 50, -10],
    'g8': [-300, 0, -10],
    'h1': [-350, 350, -10],
    'h2': [-350, 300, -10],
    'h3': [-350, 250, -10],
    'h4': [-350, 200, -10],
    'h5': [-350, 150, -10],
    'h6': [-350, 100, -10],
    'h7': [-350, 50, -10],
    'h8': [-350, 0, -10],
}

def move_to_square(square):
    if square in grid_coordinates:
        target_pose = transl(*grid_coordinates[square])
        item.setPose(target_pose)  # Set the robot's pose directly
    else:
        print(f"Square {square} not found in the grid_coordinates dictionary.")

def stockfish_move(board):
    chess.engine.SimpleEngine.popen_uci("C:/Users/dancr/chess-robot/stockfishstockfish-windows-x86-64-avx2")
    result = engine.play(board, chess.engine.Limit(time=2.0))
    return result.move

#def main():
    # Specify the full path to your Stockfish executable
    #engine_path = ("C:\Users\dancr\chess-robor\stockfish\stockfish-windows-x86-64-avx2")

    # Create a Chess engine with Stockfish
    #engine = chess.engine.SimpleEngine.popen_uci(engine_path)

    board = chess.Board()
# Loop to keep asking for input
while True:
    target_square = input("Enter the target square (e.g., a1, b3, h8) or 'no' to exit: ")

    if target_square.lower() == 'no':
        print("Exiting the program.")
        break  # Exit the loop if the user enters 'no'

    move_to_square(target_square)
    #tool.AttachClosest(list_objects=[obj])
    tool.RDK().RunProgram('Prog7')
    target_square = input("Enter the target square (e.g., a1, b3, h8) or 'no' to exit: ")

    if target_square.lower() == 'no':
        print("Exiting the program.")
        break  # Exit the loop if the user enters 'no'

    move_to_square(target_square)
    tool.RDK().RunProgram('Prog8')

    #board = chess.Board()
    #opponent_move = stockfish_move(board)
    #print("Opponent's move:", opponent_move.uci())

    # Assuming opponent_move.uci() returns a valid square (e.g., "e2e4")
    #move_to_square(opponent_move.uci())

--- Python program Prog31 ---
# Type help("robodk.robolink") or help("robodk.robomath") for more information
# Press F5 to run the script
# Documentation: https://robodk.com/doc/en/RoboDK-API.html
# Reference:     https://robodk.com/doc/en/PythonAPI/robodk.html
# Note: It is not required to keep a copy of this file, your Python script is saved with your RDK project

# You can also use the new version of the API:
from robodk import robolink    # RoboDK API
from robodk import robomath    # Robot toolbox
RDK = robolink.Robolink()

# Forward and backwards compatible use of the RoboDK API:
# Remove these 2 lines to follow python programming guidelines
from robodk import *      # RoboDK API
from robolink import *    # Robot toolbox
# Link to RoboDK
# RDK = Robolink()

# Notify user:
print('To edit this program:\nright click on the Python program, then, select "Edit Python script"')

# Program example:
item = RDK.Item('base')
if item.Valid():
    print('Item selected: ' + item.Name())
    print('Item posistion: ' + repr(item.Pose()))

#print('Items in the station:')
itemlist = RDK.ItemList()
#print(itemlist)

# Provoking an exception will display the console output if you run this script from RoboDK
#raise Exception('Program not edited.')

import tkinter as tk
import chess.engine
from robodk import robolink, transl

# RoboDK initialization
RDK = robolink.Robolink()
item = RDK.Item('My Mechanism')
tool = RDK.Item('AGV')

# Define the grid and corresponding coordinates
grid_coordinates = {
    'a1': [0, 350, -10],
    'a2': [0, 300, -10],
    'a3': [0, 250, -10],
    'a4': [0, 200, -10],
    'a5': [0, 150, -10],
    'a6': [0, 100, -10],
    'a7': [0, 50, -10],
    'a8': [0, 0, -10],
    'b1': [-50, 350, -10],
    'b2': [-50, 300, -10],
    'b3': [-50, 250, -10],
    'b4': [-50, 200, -10],
    'b5': [-50, 150, -10],
    'b6': [-50, 100, -10],
    'b7': [-50, 50, -10],
    'b8': [-50, 0, -10],
    'c1': [-100, 350, -10],
    'c2': [-100, 300, -10],
    'c3': [-100, 250, -10],
    'c4': [-100, 200, -10],
    'c5': [-100, 150, -10],
    'c6': [-100, 100, -10],
    'c7': [-100, 50, -10],
    'c8': [-100, 0, -10],
    'd1': [-150, 350, -10],
    'd2': [-150, 300, -10],
    'd3': [-150, 250, -10],
    'd4': [-150, 200, -10],
    'd5': [-150, 150, -10],
    'd6': [-150, 100, -10],
    'd7': [-150, 50, -10],
    'd8': [-150, 0, -10],
    'e1': [-200, 350, -10],
    'e2': [-200, 300, -10],
    'e3': [-200, 250, -10],
    'e4': [-200, 200, -10],
    'e5': [-200, 150, -10],
    'e6': [-200, 100, -10],
    'e7': [-200, 50, -10],
    'e8': [-200, 0, -10],
    'f1': [-250, 350, -10],
    'f2': [-250, 300, -10],
    'f3': [-250, 250, -10],
    'f4': [-250, 200, -10],
    'f5': [-250, 150, -10],
    'f6': [-250, 100, -10],
    'f7': [-250, 50, -10],
    'f8': [-250, 0, -10],
    'g1': [-300, 350, -10],
    'g2': [-300, 300, -10],
    'g3': [-300, 250, -10],
    'g4': [-300, 200, -10],
    'g5': [-300, 150, -10],
    'g6': [-300, 100, -10],
    'g7': [-300, 50, -10],
    'g8': [-300, 0, -10],
    'h1': [-350, 350, -10],
    'h2': [-350, 300, -10],
    'h3': [-350, 250, -10],
    'h4': [-350, 200, -10],
    'h5': [-350, 150, -10],
    'h6': [-350, 100, -10],
    'h7': [-350, 50, -10],
    'h8': [-350, 0, -10],
}

def move_to_square(square):
    if square in grid_coordinates:
        target_pose = transl(*grid_coordinates[square])
        item.setPose(target_pose)  # Set the robot's pose directly
    else:
        print(f"Square {square} not found in the grid_coordinates dictionary.")

def on_square_click(square):
    move_to_square(square)
    tool.RDK().RunProgram('Prog7')
    target_square = input("Enter the target square (e.g., a1, b3, h8) or 'no' to exit: ")
    if target_square.lower() == 'no':
        print("Exiting the program.")
        return  # Exit the function if the user enters 'no'
    move_to_square(target_square)
    tool.RDK().RunProgram('Prog8')

def create_button(root, row, col, square):
    button = tk.Button(root, text=square, width=3, height=1, command=lambda: on_square_click(square))
    button.grid(row=row, column=col, padx=2, pady=2)

root = tk.Tk()
root.title("Chessboard")

# Create 8x8 grid of buttons
for row in range(8):
    for col in range(8):
        square = chr(ord('a') + col) + str(8 - row)
        create_button(root, row, col, square)

root.mainloop()

--- Python program Prog32 ---
# Type help("robodk.robolink") or help("robodk.robomath") for more information
# Press F5 to run the script
# Documentation: https://robodk.com/doc/en/RoboDK-API.html
# Reference:     https://robodk.com/doc/en/PythonAPI/robodk.html
# Note: It is not required to keep a copy of this file, your Python script is saved with your RDK project

# You can also use the new version of the API:
from robodk import robolink    # RoboDK API
from robodk import robomath    # Robot toolbox
RDK = robolink.Robolink()

# Forward and backwards compatible use of the RoboDK API:
# Remove these 2 lines to follow python programming guidelines
from robodk import *      # RoboDK API
from robolink import *    # Robot toolbox
# Link to RoboDK
# RDK = Robolink()

# Notify user:
print('To edit this program:\nright click on the Python program, then, select "Edit Python script"')

# Program example:
item = RDK.Item('base')
if item.Valid():
    print('Item selected: ' + item.Name())
    print('Item posistion: ' + repr(item.Pose()))

#print('Items in the station:')
itemlist = RDK.ItemList()
#print(itemlist)

# Provoking an exception will display the console output if you run this script from RoboDK
#raise Exception('Program not edited.')
import chess
import random
from robodk import robolink, transl

# Initialize RoboDK
RDK = robolink.Robolink()
item = RDK.Item('My Mechanism')
tool = RDK.Item('AGV')

# Define the grid and corresponding coordinates
grid_coordinates = {
    'a1': [0, 350, -10],
    'a2': [0, 300, -10],
    'a3': [0, 250, -10],
    'a4': [0, 200, -10],
    'a5': [0, 150, -10],
    'a6': [0, 100, -10],
    'a7': [0, 50, -10],
    'a8': [0, 0, -10],
    'b1': [-50, 350, -10],
    'b2': [-50, 300, -10],
    'b3': [-50, 250, -10],
    'b4': [-50, 200, -10],
    'b5': [-50, 150, -10],
    'b6': [-50, 100, -10],
    'b7': [-50, 50, -10],
    'b8': [-50, 0, -10],
    'c1': [-100, 350, -10],
    'c2': [-100, 300, -10],
    'c3': [-100, 250, -10],
    'c4': [-100, 200, -10],
    'c5': [-100, 150, -10],
    'c6': [-100, 100, -10],
    'c7': [-100, 50, -10],
    'c8': [-100, 0, -10],
    'd1': [-150, 350, -10],
    'd2': [-150, 300, -10],
    'd3': [-150, 250, -10],
    'd4': [-150, 200, -10],
    'd5': [-150, 150, -10],
    'd6': [-150, 100, -10],
    'd7': [-150, 50, -10],
    'd8': [-150, 0, -10],
    'e1': [-200, 350, -10],
    'e2': [-200, 300, -10],
    'e3': [-200, 250, -10],
    'e4': [-200, 200, -10],
    'e5': [-200, 150, -10],
    'e6': [-200, 100, -10],
    'e7': [-200, 50, -10],
    'e8': [-200, 0, -10],
    'f1': [-250, 350, -10],
    'f2': [-250, 300, -10],
    'f3': [-250, 250, -10],
    'f4': [-250, 200, -10],
    'f5': [-250, 150, -10],
    'f6': [-250, 100, -10],
    'f7': [-250, 50, -10],
    'f8': [-250, 0, -10],
    'g1': [-300, 350, -10],
    'g2': [-300, 300, -10],
    'g3': [-300, 250, -10],
    'g4': [-300, 200, -10],
    'g5': [-300, 150, -10],
    'g6': [-300, 100, -10],
    'g7': [-300, 50, -10],
    'g8': [-300, 0, -10],
    'h1': [-350, 350, -10],
    'h2': [-350, 300, -10],
    'h3': [-350, 250, -10],
    'h4': [-350, 200, -10],
    'h5': [-350, 150, -10],
    'h6': [-350, 100, -10],
    'h7': [-350, 50, -10],
    'h8': [-350, 0, -10],
}

def move_to_square(square):
    if square in grid_coordinates:
        target_pose = transl(*grid_coordinates[square])
        item.setPose(target_pose)  # Set the robot's pose directly
    else:
        print(f"Square {square} not found in the grid_coordinates dictionary.")

# Create a chess board object
board = chess.Board()

# Game loop
# Game loop
# Game loop
# Game loop
# Game loop
# Game loop
while True:
    # User's move
    user_move = input("Enter your move in UCI notation (e.g., 'e2e4') or 'no' to exit: ")
    if user_move.lower() == 'no':
        print("Exiting the program.")
        break  # Exit the loop if the user enters 'no'

    move_to_square(user_move[:2])
    tool.RDK().RunProgram('Prog7')
    move_to_square(user_move[2:])
    tool.RDK().RunProgram('Prog8')

    # Print the board after the user's move
    print(board)

    # Check if the game is over after the user's move
    if board.is_game_over():
        print("Game over!")
        break

    # System's move
    legal_moves = list(board.legal_moves)
    system_move = random.choice(legal_moves)
    while system_move.uci() == user_move:
        system_move = random.choice(legal_moves)
    print("System's move:", system_move.uci())

    # Push the system's move to the board
    board.push(system_move)

    move_from = chess.square_name(system_move.from_square)
    move_to = chess.square_name(system_move.to_square)
    move_to_square(move_from)
    tool.RDK().RunProgram('Prog7')
    move_to_square(move_to)
    tool.RDK().RunProgram('Prog8')

    # Print the board after the system's move
    print(board)

    # Check if the game is over after the system's move
    if board.is_game_over():
        print("Game over!")
        break

--- Python program Prog33 ---
# Type help("robodk.robolink") or help("robodk.robomath") for more information
# Press F5 to run the script
# Documentation: https://robodk.com/doc/en/RoboDK-API.html
# Reference:     https://robodk.com/doc/en/PythonAPI/robodk.html
# Note: It is not required to keep a copy of this file, your Python script is saved with your RDK project

# You can also use the new version of the API:
from robodk import robolink    # RoboDK API
from robodk import robomath    # Robot toolbox
RDK = robolink.Robolink()

# Forward and backwards compatible use of the RoboDK API:
# Remove these 2 lines to follow python programming guidelines
from robodk import *      # RoboDK API
from robolink import *    # Robot toolbox
# Link to RoboDK
# RDK = Robolink()

# Notify user:
#print('To edit this program:\nright click on the Python program, then, select "Edit Python script"')

# Program example:


#print('Items in the station:')

#print(itemlist)

# Provoking an exception will display the console output if you run this script from RoboDK
#raise Exception('Program not edited.')
import chess
import random
from robodk import robolink, transl

# Initialize RoboDK
RDK = robolink.Robolink()
item = RDK.Item('My Mechanism')
tool = RDK.Item('AGV')

# Define the grid and corresponding coordinates
grid_coordinates = {
    'a1': [0, 350, -10],
    'a2': [0, 300, -10],
    'a3': [0, 250, -10],
    'a4': [0, 200, -10],
    'a5': [0, 150, -10],
    'a6': [0, 100, -10],
    'a7': [0, 50, -10],
    'a8': [0, 0, -10],
    'b1': [-50, 350, -10],
    'b2': [-50, 300, -10],
    'b3': [-50, 250, -10],
    'b4': [-50, 200, -10],
    'b5': [-50, 150, -10],
    'b6': [-50, 100, -10],
    'b7': [-50, 50, -10],
    'b8': [-50, 0, -10],
    'c1': [-100, 350, -10],
    'c2': [-100, 300, -10],
    'c3': [-100, 250, -10],
    'c4': [-100, 200, -10],
    'c5': [-100, 150, -10],
    'c6': [-100, 100, -10],
    'c7': [-100, 50, -10],
    'c8': [-100, 0, -10],
    'd1': [-150, 350, -10],
    'd2': [-150, 300, -10],
    'd3': [-150, 250, -10],
    'd4': [-150, 200, -10],
    'd5': [-150, 150, -10],
    'd6': [-150, 100, -10],
    'd7': [-150, 50, -10],
    'd8': [-150, 0, -10],
    'e1': [-200, 350, -10],
    'e2': [-200, 300, -10],
    'e3': [-200, 250, -10],
    'e4': [-200, 200, -10],
    'e5': [-200, 150, -10],
    'e6': [-200, 100, -10],
    'e7': [-200, 50, -10],
    'e8': [-200, 0, -10],
    'f1': [-250, 350, -10],
    'f2': [-250, 300, -10],
    'f3': [-250, 250, -10],
    'f4': [-250, 200, -10],
    'f5': [-250, 150, -10],
    'f6': [-250, 100, -10],
    'f7': [-250, 50, -10],
    'f8': [-250, 0, -10],
    'g1': [-300, 350, -10],
    'g2': [-300, 300, -10],
    'g3': [-300, 250, -10],
    'g4': [-300, 200, -10],
    'g5': [-300, 150, -10],
    'g6': [-300, 100, -10],
    'g7': [-300, 50, -10],
    'g8': [-300, 0, -10],
    'h1': [-350, 350, -10],
    'h2': [-350, 300, -10],
    'h3': [-350, 250, -10],
    'h4': [-350, 200, -10],
    'h5': [-350, 150, -10],
    'h6': [-350, 100, -10],
    'h7': [-350, 50, -10],
    'h8': [-350, 0, -10],
}

def move_to_square(square):
    if square in grid_coordinates:
        target_pose = transl(*grid_coordinates[square])
        item.setPose(target_pose)  # Set the robot's pose directly
    else:
        print(f"Square {square} not found in the grid_coordinates dictionary.")

# Create a chess board object
board = chess.Board()

# Game loop
while not board.is_game_over():
    # User's move
    user_move = input("Enter your move in UCI notation (e.g., 'e2e4'): ")
    while chess.Move.from_uci(user_move) not in board.legal_moves:
        print("Illegal move! Please enter a valid move.")
        user_move = input("Enter your move in UCI notation (e.g., 'e2e4'): ")
    board.push_uci(user_move)

    # Check if the game is over after the user's move
    if board.is_game_over():
        print("Game over!")
        break

    # Print the board after the user's move
    print("Board after your move:")
    print(board)

    # System's move
    system_move = random.choice(list(board.legal_moves))
    board.push(system_move)

    # Print the system's move in UCI notation
    print("System's move:", system_move.uci())

    # Check if the game is over after the system's move
    if board.is_game_over():
        print("Game over!")
        break

    # Print the board after the system's move
    print("Board after system's move:")
    print(board)

--- Python program Prog34 ---
# Type help("robodk.robolink") or help("robodk.robomath") for more information
# Press F5 to run the script
# Documentation: https://robodk.com/doc/en/RoboDK-API.html
# Reference:     https://robodk.com/doc/en/PythonAPI/robodk.html
# Note: It is not required to keep a copy of this file, your Python script is saved with your RDK project

# You can also use the new version of the API:
from robodk import robolink    # RoboDK API
from robodk import robomath    # Robot toolbox
RDK = robolink.Robolink()

# Forward and backwards compatible use of the RoboDK API:
# Remove these 2 lines to follow python programming guidelines
from robodk import *      # RoboDK API
from robolink import *    # Robot toolbox
# Link to RoboDK
# RDK = Robolink()

import chess
import random
from robodk import robolink, transl

# Initialize RoboDK
RDK = robolink.Robolink()
item = RDK.Item('My Mechanism')
tool = RDK.Item('AGV')

# Define the grid and corresponding coordinates
grid_coordinates = {
    'a1': [0, 350, -10],
    'a2': [0, 300, -10],
    'a3': [0, 250, -10],
    'a4': [0, 200, -10],
    'a5': [0, 150, -10],
    'a6': [0, 100, -10],
    'a7': [0, 50, -10],
    'a8': [0, 0, -10],
    'b1': [-50, 350, -10],
    'b2': [-50, 300, -10],
    'b3': [-50, 250, -10],
    'b4': [-50, 200, -10],
    'b5': [-50, 150, -10],
    'b6': [-50, 100, -10],
    'b7': [-50, 50, -10],
    'b8': [-50, 0, -10],
    'c1': [-100, 350, -10],
    'c2': [-100, 300, -10],
    'c3': [-100, 250, -10],
    'c4': [-100, 200, -10],
    'c5': [-100, 150, -10],
    'c6': [-100, 100, -10],
    'c7': [-100, 50, -10],
    'c8': [-100, 0, -10],
    'd1': [-150, 350, -10],
    'd2': [-150, 300, -10],
    'd3': [-150, 250, -10],
    'd4': [-150, 200, -10],
    'd5': [-150, 150, -10],
    'd6': [-150, 100, -10],
    'd7': [-150, 50, -10],
    'd8': [-150, 0, -10],
    'e1': [-200, 350, -10],
    'e2': [-200, 300, -10],
    'e3': [-200, 250, -10],
    'e4': [-200, 200, -10],
    'e5': [-200, 150, -10],
    'e6': [-200, 100, -10],
    'e7': [-200, 50, -10],
    'e8': [-200, 0, -10],
    'f1': [-250, 350, -10],
    'f2': [-250, 300, -10],
    'f3': [-250, 250, -10],
    'f4': [-250, 200, -10],
    'f5': [-250, 150, -10],
    'f6': [-250, 100, -10],
    'f7': [-250, 50, -10],
    'f8': [-250, 0, -10],
    'g1': [-300, 350, -10],
    'g2': [-300, 300, -10],
    'g3': [-300, 250, -10],
    'g4': [-300, 200, -10],
    'g5': [-300, 150, -10],
    'g6': [-300, 100, -10],
    'g7': [-300, 50, -10],
    'g8': [-300, 0, -10],
    'h1': [-350, 350, -10],
    'h2': [-350, 300, -10],
    'h3': [-350, 250, -10],
    'h4': [-350, 200, -10],
    'h5': [-350, 150, -10],
    'h6': [-350, 100, -10],
    'h7': [-350, 50, -10],
    'h8': [-350, 0, -10],
}

def move_to_square(square):
    if square in grid_coordinates:
        target_pose = transl(*grid_coordinates[square])
        item.setPose(target_pose)  # Set the robot's pose directly
    else:
        print(f"Square {square} not found in the grid_coordinates dictionary.")

# Create a chess board object
board = chess.Board()

# Game loop
while not board.is_game_over():
    # User's move
    user_move = input("Enter your move in UCI notation (e.g., 'e2e4'): ")
    while chess.Move.from_uci(user_move) not in board.legal_moves:
        print("Illegal move! Please enter a valid move.")
        user_move = input("Enter your move in UCI notation (e.g., 'e2e4'): ")
    board.push_uci(user_move)
    move_to_square(user_move[:2])
    move_to_square(user_move[2:])

    # Check if the game is over after the user's move
    if board.is_game_over():
        print("Game over!")
        break

    # Print the board after the user's move
    print("Board after your move:")
    print(board)

    # System's move
    system_move = random.choice(list(board.legal_moves))
    board.push(system_move)
    move_to_square(chess.square_name(system_move.from_square))
    move_to_square(chess.square_name(system_move.to_square))

    # Print the system's move in UCI notation
    print("System's move:", system_move.uci())

    # Check if the game is over after the system's move
    if board.is_game_over():
        print("Game over!")
        break

    # Print the board after the system's move
    print("Board after system's move:")
    print(board)

--- Python program Prog35 ---
# Type help("robodk.robolink") or help("robodk.robomath") for more information
# Press F5 to run the script
# Documentation: https://robodk.com/doc/en/RoboDK-API.html
# Reference:     https://robodk.com/doc/en/PythonAPI/robodk.html
# Note: It is not required to keep a copy of this file, your Python script is saved with your RDK project

# You can also use the new version of the API:
from robodk import robolink    # RoboDK API
from robodk import robomath    # Robot toolbox
RDK = robolink.Robolink()

# Forward and backwards compatible use of the RoboDK API:
# Remove these 2 lines to follow python programming guidelines
from robodk import *      # RoboDK API
from robolink import *    # Robot toolbox
# Link to RoboDK
# RDK = Robolink()


import chess
import random
from robodk import robolink, transl

# Initialize RoboDK
RDK = robolink.Robolink()
item = RDK.Item('My Mechanism')
tool = RDK.Item('AGV')

# Define the grid and corresponding coordinates
grid_coordinates = {
    'a1': [0, 350, -10],
    'a2': [0, 300, -10],
    'a3': [0, 250, -10],
    'a4': [0, 200, -10],
    'a5': [0, 150, -10],
    'a6': [0, 100, -10],
    'a7': [0, 50, -10],
    'a8': [0, 0, -10],
    'b1': [-50, 350, -10],
    'b2': [-50, 300, -10],
    'b3': [-50, 250, -10],
    'b4': [-50, 200, -10],
    'b5': [-50, 150, -10],
    'b6': [-50, 100, -10],
    'b7': [-50, 50, -10],
    'b8': [-50, 0, -10],
    'c1': [-100, 350, -10],
    'c2': [-100, 300, -10],
    'c3': [-100, 250, -10],
    'c4': [-100, 200, -10],
    'c5': [-100, 150, -10],
    'c6': [-100, 100, -10],
    'c7': [-100, 50, -10],
    'c8': [-100, 0, -10],
    'd1': [-150, 350, -10],
    'd2': [-150, 300, -10],
    'd3': [-150, 250, -10],
    'd4': [-150, 200, -10],
    'd5': [-150, 150, -10],
    'd6': [-150, 100, -10],
    'd7': [-150, 50, -10],
    'd8': [-150, 0, -10],
    'e1': [-200, 350, -10],
    'e2': [-200, 300, -10],
    'e3': [-200, 250, -10],
    'e4': [-200, 200, -10],
    'e5': [-200, 150, -10],
    'e6': [-200, 100, -10],
    'e7': [-200, 50, -10],
    'e8': [-200, 0, -10],
    'f1': [-250, 350, -10],
    'f2': [-250, 300, -10],
    'f3': [-250, 250, -10],
    'f4': [-250, 200, -10],
    'f5': [-250, 150, -10],
    'f6': [-250, 100, -10],
    'f7': [-250, 50, -10],
    'f8': [-250, 0, -10],
    'g1': [-300, 350, -10],
    'g2': [-300, 300, -10],
    'g3': [-300, 250, -10],
    'g4': [-300, 200, -10],
    'g5': [-300, 150, -10],
    'g6': [-300, 100, -10],
    'g7': [-300, 50, -10],
    'g8': [-300, 0, -10],
    'h1': [-350, 350, -10],
    'h2': [-350, 300, -10],
    'h3': [-350, 250, -10],
    'h4': [-350, 200, -10],
    'h5': [-350, 150, -10],
    'h6': [-350, 100, -10],
    'h7': [-350, 50, -10],
    'h8': [-350, 0, -10],
}

def move_to_square(square):
    if square in grid_coordinates:
        target_pose = transl(*grid_coordinates[square])
        item.setPose(target_pose)  # Set the robot's pose directly
        print(f"Robot moves to square {square}")
    else:
        print(f"Square {square} not found in the grid_coordinates dictionary.")

# Create a chess board object
board = chess.Board()

# Game loop
while not board.is_game_over():
    # User's move
    user_move = input("Enter your move in UCI notation (e.g., 'e2e4'): ")
    while chess.Move.from_uci(user_move) not in board.legal_moves:
        print("Illegal move! Please enter a valid move.")
        user_move = input("Enter your move in UCI notation (e.g., 'e2e4'): ")
    board.push_uci(user_move)
    move_to_square(user_move[:2])
    move_to_square(user_move[2:])

    # Check if the game is over after the user's move
    if board.is_game_over():
        print("Game over!")
        break

    # Print the board after the user's move
    print("Board after your move:")
    print(board)

    # System's move
    system_move = random.choice(list(board.legal_moves))
    board.push(system_move)
    move_to_square(chess.square_name(system_move.from_square))
    move_to_square(chess.square_name(system_move.to_square))

    # Print the system's move in UCI notation
    print("System's move:", system_move.uci())

    # Check if the game is over after the system's move
    if board.is_game_over():
        print("Game over!")
        break

    # Print the board after the system's move
    print("Board after system's move:")
    print(board)

--- Python program Prog36 ---
# Type help("robodk.robolink") or help("robodk.robomath") for more information
# Press F5 to run the script
# Documentation: https://robodk.com/doc/en/RoboDK-API.html
# Reference:     https://robodk.com/doc/en/PythonAPI/robodk.html
# Note: It is not required to keep a copy of this file, your Python script is saved with your RDK project

# You can also use the new version of the API:
from robodk import robolink    # RoboDK API
from robodk import robomath    # Robot toolbox
RDK = robolink.Robolink()

# Forward and backwards compatible use of the RoboDK API:
# Remove these 2 lines to follow python programming guidelines
from robodk import *      # RoboDK API
from robolink import *    # Robot toolbox
import chess
import random
from stockfish import Stockfish

# Initialize Stockfish engine
stockfish = Stockfish("C:/Users/dancr/chess-robot/stockfish/stockfish-windows-x86-64-avx2.exe")

# Set Stockfish parameters (optional)
stockfish.set_depth(10)  # Adjust the search depth
stockfish.set_skill_level(20)  # Adjust the skill level

# Create a chess board object
board = chess.Board()

# Game loop
while not board.is_game_over():
    # User's move
    user_move = input("Enter your move in UCI notation (e.g., 'e2e4'): ")
    while chess.Move.from_uci(user_move) not in board.legal_moves:
        print("Illegal move! Please enter a valid move.")
        user_move = input("Enter your move in UCI notation (e.g., 'e2e4'): ")
    board.push_uci(user_move)

    # Check if the game is over after the user's move
    if board.is_game_over():
        print("Game over!")
        break

    # Print the board after the user's move
    print("Board after your move:")
    print(board)

    # System's move
    stockfish.set_fen_position(board.fen())  # Set the board position for Stockfish
    system_move = stockfish.get_best_move()
    print("Stockfish suggests move:", system_move)
    board.push(chess.Move.from_uci(system_move))

    # Print the system's move in UCI notation
    print("System's move:", system_move)

    # Check if the game is over after the system's move
    if board.is_game_over():
        print("Game over!")
        break

    # Print the board after the system's move
    print("Board after system's move:")
    print(board)

--- Python program final ---
# Type help("robodk.robolink") or help("robodk.robomath") for more information
# Press F5 to run the script
# Documentation: https://robodk.com/doc/en/RoboDK-API.html
# Reference:     https://robodk.com/doc/en/PythonAPI/robodk.html
# Note: It is not required to keep a copy of this file, your Python script is saved with your RDK project

# You can also use the new version of the API:
from robodk import robolink    # RoboDK API
from robodk import robomath    # Robot toolbox
RDK = robolink.Robolink()

# Forward and backwards compatible use of the RoboDK API:
# Remove these 2 lines to follow python programming guidelines
from robodk import *      # RoboDK API
from robolink import *    # Robot toolbox
# Link to RoboDK
# RDK = Robolink()

import chess
import random
from stockfish import Stockfish

# Initialize Stockfish engine
stockfish = Stockfish("C:/Users/dancr/chess-robot/stockfish/stockfish-windows-x86-64-avx2.exe")#   Replace with the actual path

# Define the grid and corresponding coordinates
grid_coordinates = {
    'a1': [0, 350, -10],
    'a2': [0, 300, -10],
    'a3': [0, 250, -10],
    'a4': [0, 200, -10],
    'a5': [0, 150, -10],
    'a6': [0, 100, -10],
    'a7': [0, 50, -10],
    'a8': [0, 0, -10],
    'b1': [-50, 350, -10],
    'b2': [-50, 300, -10],
    'b3': [-50, 250, -10],
    'b4': [-50, 200, -10],
    'b5': [-50, 150, -10],
    'b6': [-50, 100, -10],
    'b7': [-50, 50, -10],
    'b8': [-50, 0, -10],
    'c1': [-100, 350, -10],
    'c2': [-100, 300, -10],
    'c3': [-100, 250, -10],
    'c4': [-100, 200, -10],
    'c5': [-100, 150, -10],
    'c6': [-100, 100, -10],
    'c7': [-100, 50, -10],
    'c8': [-100, 0, -10],
    'd1': [-150, 350, -10],
    'd2': [-150, 300, -10],
    'd3': [-150, 250, -10],
    'd4': [-150, 200, -10],
    'd5': [-150, 150, -10],
    'd6': [-150, 100, -10],
    'd7': [-150, 50, -10],
    'd8': [-150, 0, -10],
    'e1': [-200, 350, -10],
    'e2': [-200, 300, -10],
    'e3': [-200, 250, -10],
    'e4': [-200, 200, -10],
    'e5': [-200, 150, -10],
    'e6': [-200, 100, -10],
    'e7': [-200, 50, -10],
    'e8': [-200, 0, -10],
    'f1': [-250, 350, -10],
    'f2': [-250, 300, -10],
    'f3': [-250, 250, -10],
    'f4': [-250, 200, -10],
    'f5': [-250, 150, -10],
    'f6': [-250, 100, -10],
    'f7': [-250, 50, -10],
    'f8': [-250, 0, -10],
    'g1': [-300, 350, -10],
    'g2': [-300, 300, -10],
    'g3': [-300, 250, -10],
    'g4': [-300, 200, -10],
    'g5': [-300, 150, -10],
    'g6': [-300, 100, -10],
    'g7': [-300, 50, -10],
    'g8': [-300, 0, -10],
    'h1': [-350, 350, -10],
    'h2': [-350, 300, -10],
    'h3': [-350, 250, -10],
    'h4': [-350, 200, -10],
    'h5': [-350, 150, -10],
    'h6': [-350, 100, -10],
    'h7': [-350, 50, -10],
    'h8': [-350, 0, -10],
}

# Function to move the robot to a specific square
def move_to_square(square):
    if square in grid_coordinates:
        target_pose = grid_coordinates[square]
        print(f"Robot moves to square {square}: {target_pose}")
        # Add your robot movement logic here to move the robot to the target_pose
    else:
        print(f"Square {square} not found in the grid_coordinates dictionary.")

# Create a chess board object
board = chess.Board()

# Game loop
while not board.is_game_over():
    # User's move
    user_move = input("Enter your move in UCI notation (e.g., 'e2e4'): ")
    while chess.Move.from_uci(user_move) not in board.legal_moves:
        print("Illegal move! Please enter a valid move.")
        user_move = input("Enter your move in UCI notation (e.g., 'e2e4'): ")
    board.push_uci(user_move)

    # Check if the game is over after the user's move
    if board.is_game_over():
        print("Game over!")
        break

    # Print the board after the user's move
    print("Board after your move:")
    print(board)

    # System's move
    stockfish.set_fen_position(board.fen())  # Set the board position for Stockfish
    system_move = stockfish.get_best_move()
    print("Stockfish suggests move:", system_move)

    # Convert Stockfish's move to square coordinates
    from_square = system_move[:2]

    to_square = system_move[2:]

    # Move the robot to the 'from' square
    move_to_square(from_square)
    print(move_to_square(from_square))
    # Make the robot pick up the piece from the 'from' square (if necessary)
    # Add your code to handle the robot picking up the piece here

    # Move the robot to the 'to' square
    move_to_square(to_square)
    print(move_to_square(to_square))
    # Make the robot drop the piece at the 'to' square (if necessary)
    # Add your code to handle the robot dropping the piece here

    # Push the move to the board
    board.push(chess.Move.from_uci(system_move))

    # Print the board after the system's move
    print("Board after system's move:")
    print(board)

--- Python program stockfish ---
# Type help("robodk.robolink") or help("robodk.robomath") for more information
# Press F5 to run the script
# Documentation: https://robodk.com/doc/en/RoboDK-API.html
# Reference:     https://robodk.com/doc/en/PythonAPI/robodk.html
# Note: It is not required to keep a copy of this file, your Python script is saved with your RDK project

# You can also use the new version of the API:
from robodk import robolink    # RoboDK API
from robodk import robomath    # Robot toolbox
RDK = robolink.Robolink()

# Forward and backwards compatible use of the RoboDK API:
# Remove these 2 lines to follow python programming guidelines
from robodk import *      # RoboDK API
from robolink import *    # Robot toolbox
# Link to RoboDK
# RDK = Robolink()
item = RDK.Item('My Mechanism')
tool = RDK.Item('AGV')
if item.Valid():
    print('Item selected: ' + item.Name())
    print('Item position before move: ' + repr(item.Pose()))

import chess
import random
from stockfish import Stockfish

# Initialize Stockfish engine
stockfish = Stockfish("C:/Users/dancr/chess-robot/stockfish/stockfish-windows-x86-64-avx2.exe")  # Replace with the actual path

# Define the grid and corresponding coordinates
grid_coordinates = {

    'a1': [0, 350, -10],
    'a2': [0, 300, -10],
    'a3': [0, 250, -10],
    'a4': [0, 200, -10],
    'a5': [0, 150, -10],
    'a6': [0, 100, -10],
    'a7': [0, 50, -10],
    'a8': [0, 0, -10],
    'b1': [-50, 350, -10],
    'b2': [-50, 300, -10],
    'b3': [-50, 250, -10],
    'b4': [-50, 200, -10],
    'b5': [-50, 150, -10],
    'b6': [-50, 100, -10],
    'b7': [-50, 50, -10],
    'b8': [-50, 0, -10],
    'c1': [-100, 350, -10],
    'c2': [-100, 300, -10],
    'c3': [-100, 250, -10],
    'c4': [-100, 200, -10],
    'c5': [-100, 150, -10],
    'c6': [-100, 100, -10],
    'c7': [-100, 50, -10],
    'c8': [-100, 0, -10],
    'd1': [-150, 350, -10],
    'd2': [-150, 300, -10],
    'd3': [-150, 250, -10],
    'd4': [-150, 200, -10],
    'd5': [-150, 150, -10],
    'd6': [-150, 100, -10],
    'd7': [-150, 50, -10],
    'd8': [-150, 0, -10],
    'e1': [-200, 350, -10],
    'e2': [-200, 300, -10],
    'e3': [-200, 250, -10],
    'e4': [-200, 200, -10],
    'e5': [-200, 150, -10],
    'e6': [-200, 100, -10],
    'e7': [-200, 50, -10],
    'e8': [-200, 0, -10],
    'f1': [-250, 350, -10],
    'f2': [-250, 300, -10],
    'f3': [-250, 250, -10],
    'f4': [-250, 200, -10],
    'f5': [-250, 150, -10],
    'f6': [-250, 100, -10],
    'f7': [-250, 50, -10],
    'f8': [-250, 0, -10],
    'g1': [-300, 350, -10],
    'g2': [-300, 300, -10],
    'g3': [-300, 250, -10],
    'g4': [-300, 200, -10],
    'g5': [-300, 150, -10],
    'g6': [-300, 100, -10],
    'g7': [-300, 50, -10],
    'g8': [-300, 0, -10],
    'h1': [-350, 350, -10],
    'h2': [-350, 300, -10],
    'h3': [-350, 250, -10],
    'h4': [-350, 200, -10],
    'h5': [-350, 150, -10],
    'h6': [-350, 100, -10],
    'h7': [-350, 50, -10],
    'h8': [-350, 0, -10],

}

# Function to move the robot to a specific square
def move_from_square(from_square):
    if from_square in grid_coordinates:
        target_pose = transl(*grid_coordinates[from_square])
        item.setPose(target_pose)
        print(f"Robot moves to square {from_square}: {target_pose}")
        # Add your robot movement logic here to move the robot to the target_pose
    else:
        print(f"Square {from_square} not found in the grid_coordinates dictionary.")
def move_to_square(to_square):
    if to_square in grid_coordinates:
        target_pose = transl(*grid_coordinates[to_square])
        item.setPose(target_pose)
        print(f"Robot moves to square {to_square}: {target_pose}")
        # Add your robot movement logic here to move the robot to the target_pose
    else:
        print(f"Square {to_square} not found in the grid_coordinates dictionary.")
# Create a chess board object
board = chess.Board()

# Game loop
while not board.is_game_over():
    # User's move
    user_move = input("Enter your move in UCI notation (e.g., 'e2e4'): ")
    while chess.Move.from_uci(user_move) not in board.legal_moves:
        print("Illegal move! Please enter a valid move.")
        user_move = input("Enter your move in UCI notation (e.g., 'e2e4'): ")
    board.push_uci(user_move)

   # Convert Stockfish's move to square coordinates
    #from_square = user_move[:2]
    #to_square = user_move[2:]

    #move_from_square(from_square)
    #tool.RDK().RunProgram('Prog7')
    # Move the robot to the 'to' square
    #move_to_square(to_square)
    #tool.RDK().RunProgram('Prog8')
    # Push the move to the board

    # Check if the game is over after the user's move
    if board.is_game_over():
        print("Game over!")
        break

    # Print the board after the user's move
    print("Board after your move:")
    print(board)

    # System's move
    stockfish.set_fen_position(board.fen())  # Set the board position for Stockfish
    system_move = stockfish.get_best_move()
    print("Stockfish suggests move:", system_move)

    # Convert Stockfish's move to square coordinates
    from_square = system_move[:2]
    to_square = system_move[2:]

    # Move the robot to the 'from' square
    move_from_square(from_square)
    tool.RDK().RunProgram('Prog7')
    # Move the robot to the 'to' square
    move_to_square(to_square)
    tool.RDK().RunProgram('Prog8')
    # Push the move to the board
    board.push(chess.Move.from_uci(system_move))

    # Print the board after the system's move
    print("Board after system's move:")
    print(board)

--- Python program RoboDKChessStockfishfinal ---
# Type help("robodk.robolink") or help("robodk.robomath") for more information
# Press F5 to run the script
# Documentation: https://robodk.com/doc/en/RoboDK-API.html
# Reference:     https://robodk.com/doc/en/PythonAPI/robodk.html
# Note: It is not required to keep a copy of this file, your Python script is saved with your RDK project

# You can also use the new version of the API:
from robodk import robolink    # RoboDK API
from robodk import robomath    # Robot toolbox
RDK = robolink.Robolink()

# Forward and backwards compatible use of the RoboDK API:
# Remove these 2 lines to follow python programming guidelines
from robodk import *      # RoboDK API
from robolink import *    # Robot toolbox
# Link to RoboDK
# RDK = Robolink()

# Notify user:
print('To edit this program:\nright click on the Python program, then, select "Edit Python script"')

# Program example:

item = RDK.Item('My Mechanism')
tool = RDK.Item('microagv1')
if item.Valid():
    print('Item selected: ' + item.Name())
    print('Item position before move: ' + repr(item.Pose()))

#print('Items in the station:')
itemlist = RDK.ItemList()
#print(itemlist)

# Provoking an exception will display the console output if you run this script from RoboDK
#raise Exception('Program not edited.')
import chess
import random
from stockfish import Stockfish

# Initialize Stockfish engine
stockfish = Stockfish("C:/Users/dancr/chess-robot/stockfish/stockfish-windows-x86-64-avx2.exe")  # Replace with the actual path

# Define the grid and corresponding coordinates
grid_coordinates = {
    'a1': [0, 350, -10],
    'a2': [0, 300, -10],
    'a3': [0, 250, -10],
    'a4': [0, 200, -10],
    'a5': [0, 150, -10],
    'a6': [0, 100, -10],
    'a7': [0, 50, -10],
    'a8': [0, 0, -10],
    'b1': [-50, 350, -10],
    'b2': [-50, 300, -10],
    'b3': [-50, 250, -10],
    'b4': [-50, 200, -10],
    'b5': [-50, 150, -10],
    'b6': [-50, 100, -10],
    'b7': [-50, 50, -10],
    'b8': [-50, 0, -10],
   'c1': [-100, 350, -10],
    'c2': [-100, 300, -10],
    'c3': [-100, 250, -10],
    'c4': [-100, 200, -10],
    'c5': [-100, 150, -10],
    'c6': [-100, 100, -10],
    'c7': [-100, 50, -10],
    'c8': [-100, 0, -10],
    'd1': [-150, 350, -10],
    'd2': [-150, 300, -10],
    'd3': [-150, 250, -10],
    'd4': [-150, 200, -10],
    'd5': [-150, 150, -10],
    'd6': [-150, 100, -10],
    'd7': [-150, 50, -10],
    'd8': [-150, 0, -10],
    'e1': [-200, 350, -10],
    'e2': [-200, 300, -10],
    'e3': [-200, 250, -10],
    'e4': [-200, 200, -10],
    'e5': [-200, 150, -10],
    'e6': [-200, 100, -10],
    'e7': [-200, 50, -10],
    'e8': [-200, 0, -10],
    'f1': [-250, 350, -10],
    'f2': [-250, 300, -10],
    'f3': [-250, 250, -10],
    'f4': [-250, 200, -10],
    'f5': [-250, 150, -10],
    'f6': [-250, 100, -10],
    'f7': [-250, 50, -10],
    'f8': [-250, 0, -10],
    'g1': [-300, 350, -10],
    'g2': [-300, 300, -10],
    'g3': [-300, 250, -10],
    'g4': [-300, 200, -10],
    'g5': [-300, 150, -10],
    'g6': [-300, 100, -10],
    'g7': [-300, 50, -10],
    'g8': [-300, 0, -10],
    'h1': [-350, 350, -10],
    'h2': [-350, 300, -10],
    'h3': [-350, 250, -10],
    'h4': [-350, 200, -10],
    'h5': [-350, 150, -10],
    'h6': [-350, 100, -10],
    'h7': [-350, 50, -10],
    'h8': [-350, 0, -10],
    # Rest of the grid coordinates...
}

# Function to move the robot to a specific square from user input
def user_move_from_square(user_from_square):
    if user_from_square in grid_coordinates:
        target_pose = transl(*grid_coordinates[user_from_square])
        item.setPose(target_pose)
        print(f"Robot moves to square {user_from_square}: {target_pose}")
    else:
        print(f"Square {square} not found in the grid_coordinates dictionary.")

#def user_move_to_square(user_to_square):
    #if user_to_square in grid_coordinates:
        #target_pose = transl(*grid_coordinates[user_to_square])
        #item.setPose(target_pose)
        #print(f"Robot moves to square {user_to_square}: {target_pose}")
    #else:
        #print(f"Square {square} not found in the grid_coordinates dictionary.")

def system_move_from_square(system_from_square):
    if system_from_square in grid_coordinates:
        target_pose = transl(*grid_coordinates[system_from_square])
        item.setPose(target_pose)
        print(f"Robot moves to square {system_from_square}: {target_pose}")
    else:
        print(f"Square {square} not found in the grid_coordinates dictionary.")

#def system_move_to_square(system_to_square):
    #if system_to_square in grid_coordinates:
        #target_pose = transl(*grid_coordinates[system_to_square])
        #item.setPose(target_pose)
        #print(f"Robot moves to square {system_to_square}: {target_pose}")
    #else:
        #print(f"Square {square} not found in the grid_coordinates dictionary.")
def hide_piece_at_system_square(system_to_square):
    # Check if there is a piece at the given square and hide it if it exists
    if system_to_square in grid_coordinates:
        piece_item = RDK.Item(system_to_square)  # Assuming the name of the item representing the piece is the square name
        if piece_item.Valid():
            piece_item.setVisible(False)
            print(f"Hiding piece at square {system_to_square}")
        else:
            print(f"No piece found at square {system_to_square}")
def hide_piece_at_user_square(user_to_square):
    # Check if there is a piece at the given square and hide it if it exists
    if user_to_square in grid_coordinates:
        piece_item = RDK.Item(user_to_square)  # Assuming the name of the item representing the piece is the square name
        if piece_item.Valid():
            piece_item.setVisible(False)
            print(f"Hiding piece at square {user_to_square}")
        else:
            print(f"No piece found at square {user_to_square}")
# Function to move the robot to a specific square from user input
def user_move_to_square(user_to_square):
    if user_to_square in grid_coordinates:
        # Check if there's a piece at the target square and hide it if there is
        hide_piece_at_user_square(user_to_square)

        # Move the robot to the target square
        target_pose = transl(*grid_coordinates[user_to_square])
        item.setPose(target_pose)
        print(f"Robot moves to square {user_to_square}: {target_pose}")
    else:
        print(f"Square {user_to_square} not found in the grid_coordinates dictionary.")

# Function to move the robot to a specific square for the system's move
def system_move_to_square(system_to_square):
    if system_to_square in grid_coordinates:
        # Check if there's a piece at the target square and hide it if there is
        hide_piece_at_system_square(system_to_square)

        # Move the robot to the target square
        target_pose = transl(*grid_coordinates[system_to_square])
        item.setPose(target_pose)
        print(f"Robot moves to square {system_to_square}: {target_pose}")
    else:
        print(f"Square {system_to_square} not found in the grid_coordinates dictionary.")



# Create a chess board object
board = chess.Board()

# Game loop
while not board.is_game_over():
    # User's move
    user_move = input("Enter your move in UCI notation (e.g., 'e2e4'): ")
    while chess.Move.from_uci(user_move) not in board.legal_moves:
        print("Illegal move! Please enter a valid move.")
        user_move = input("Enter your move in UCI notation (e.g., 'e2e4'): ")
    board.push_uci(user_move)
    user_from_square = user_move[:2]
    user_to_square = user_move[2:]
    # Move the robot to the 'from' square
    user_move_from_square(user_from_square)
    tool.RDK().RunProgram('Prog7')
    # Move the robot to the 'to' square
    user_move_to_square(user_to_square)
    tool.RDK().RunProgram('Prog8')


    # Check if the game is over after the user's move
    if board.is_game_over():
        print("Game over!")
        break

    # Print the board after the user's move
    print("Board after your move:")
    print(board)

    # System's move
    stockfish.set_fen_position(board.fen())  # Set the board position for Stockfish
    system_move = stockfish.get_best_move()
    print("Stockfish suggests move:", system_move)

    # Convert Stockfish's move to square coordinates
    system_from_square = system_move[:2]
    system_to_square = system_move[2:]

    # Move the robot to the 'from' square
    system_move_from_square(system_from_square)
    tool.RDK().RunProgram('Prog7')
    # Move the robot to the 'to' square
    system_move_to_square(system_to_square)
    tool.RDK().RunProgram('Prog8')
    # Push the move to the board

    # Push the move to the board
    board.push(chess.Move.from_uci(system_move))

    # Print the board after the system's move
    print("Board after system's move:")
    print(board)
